FUNCTION_BLOCK FB_TCMultiLevelSeq EXTENDS Tc3_HBI_System.FB_Basic
VAR_INPUT
	iLevel								: UINT;
	lvlAlmMod							: ST_AlarmModules;
END_VAR
VAR_OUTPUT
END_VAR
VAR	
	// Cylinder instance
	fbTCDrawerExtRet					: Tc3_HBI_Cylinder.FB_Cylinder;
	inTCDrawerExtRet					: Tc3_HBI_Cylinder.I_Cylinder:= fbTCDrawerExtRet;
		                        		
	fbTCDrawerUpDn						: Tc3_HBI_Cylinder.FB_Cylinder;
	inTCDrawerUpDn						: Tc3_HBI_Cylinder.I_Cylinder:= fbTCDrawerUpDn;
	
	fbMotor_Ready 						: Tc3_HBI_Utilities.FB_SensorSignal;
	fbMotor_Home_Position 				: Tc3_HBI_Utilities.FB_SensorSignal;
	fbMotor_Position_Reached			: Tc3_HBI_Utilities.FB_SensorSignal;
	fbMotor_Ps_Table_Active				: Tc3_HBI_Utilities.FB_SensorSignal; //temp use for level1 movein ready
	fbMotor_Error						: Tc3_HBI_Utilities.FB_SensorSignal;
	fbBD_ipBdoor 						: Tc3_HBI_Utilities.FB_BackDoor_Digital;
	
	delay								: FB_Delay;
	
	inPOn								: BOOL;
	outPon								: BOOL;

	doorLockChkTim						: TON; // Timer To Check DoorLockFeedBack After DoorLock Output is On.
	
	DIFU								: R_TRIG;
	
	stMLVIO 							: ST_TCMultiLevel_VIO;
	stDbStnVIO							: ST_DebugStation_VIO; // For Debug Sation VIO; 
	stMLDIO 							: ST_TCMultiLevel_DIO;
	stMLBIO								: ST_TCMultiLevel_BIO;
	stTCMLSeqParam 						: ST_TCMultiLevelSeqParam;
	stTCColVIO							: ST_TCColumn_VIO;
	stTCColDIO							: ST_TCColumn_DIO;
	
	//for log purpose
	stOldMLVIO 							: ST_TCMultiLevel_VIO;
	stOldAlarm							: ST_AlarmModules;
	
	FB_M_nCyclic_tSensorDelay			: TIME	:= T#200MS; // By default
	FB_M_nCyclic_tSensorTimeOut			: TIME	:= T#10S;

	// Common var 
	bPause 								: BOOL; // Sequence pause
	bBypassSingleMove 					: BOOL	:= TRUE;
	bStep								: BOOL;
	rtStep								: R_TRIG;
	rtStepCase							: R_TRIG;
	rtError								: R_TRIG;
	iStkSeqCase 						: INT;
	iSeqStep							: INT;
	iSysRsetSeqStep						: INT;
	arrSeqStep							: ARRAY [0..50] OF E_SeqSts; // Seq
	arrSysRsetSeqStep					: ARRAY [0..50] OF E_SeqSts; // Sys Rset seq
	
	sMessage 							: STRING;
	bErrClear							: BOOL;
	bStepDone							: BOOL;
	bSafeExecute						: BOOL;
	iStkSingStackUp						: INT;
	iLibrySts 							: ARRAY [1..20] OF UDINT;
	                            		
	sMsg 								: STRING;
	FB_M_nCyclic_tDelay					: TIME	:= T#200MS;
	
	nI									: UINT;
	rtStartTrig							: R_Trig;
	rtStopTrig							: R_Trig;
	StartPbDly							: Ton;
	StopPbDly							: Ton;
	                            		
	btest								: BOOL;
	
	tDPSDelayToComplete					: TON; // DPSPowerOnOff
	tDPSDelayToAutoComplete				: TON; // DPSPowerAuto
	                            		
	tAPACPwrDelayToComplete				: TON; // AP240ACPowerOnOff
	tAPACPwrDelayToAutoComplete			: TON; // AP240ACPowerAuto
	
	tBef								: TIME; // Before Dwr Action
	tAft								: TIME; // After Dwr Action
	tSpn								: REAL; // Duration Time Span
	tUpDnlock							: BOOL;
	tInOutlock							: BOOL;
	i									: INT;
	pwrOnChkTim							: TON; // PowerOnFeedBackCheck Delay After Power On Durin SystemRset
	
	DIFUTstPresent						: R_TRIG;
	DIFUOn_TstPwr						: R_TRIG;
	DIFUAPPresent						: R_TRIG;
	DIFUOn_AP240Pwr						: R_TRIG;
	DIFUSet_bChkTstOn					: R_TRIG; 	
	DIFUSet_bChkAP240On					: R_TRIG; 	
	
	
	tstOnCheckTim						: TON; // delay to check TesterOnFeedback
	ap240OnCheckTim						: TON; // delay to check AP240OnFeedback
	tstPresentTim						: TON; // delay to On Tester Air Valve after Tester Present
	apPresentTimer						: TON;
	isLeakage							: BOOL;
	isGroundFault						: BOOL;
	isTstPwrOnFault						: BOOL;
	TBOT_TC_ACPower_Signal					: BOOL;
	bTIISenSimArray						: ARRAY[1..NO_OF_TII_SENSOR] OF BOOL;  //TII Sensor Sim by HMI
	bBtnSimArray						: ARRAY[1..NO_OF_BTNLED] OF BOOL;  //Btn Press Sim by HMI

//<TII Interlock>
	itl_opAP_240ACPwrEnable  			: BOOL	:= FALSE;
    itl_opDoorOpenReqLED				: BOOL	:= FALSE;
    itl_opAlarmLED 						: BOOL	:= FALSE;
    itl_opTesterAPDetachReqBtnLED		: BOOL	:= FALSE;
    itl_opTesterDrawerAirOffReqBtnLED   : BOOL	:= FALSE;
    itl_opAP_SafeToMoveSignal           : BOOL	:= FALSE;
    itl_opAP_TCCReset					: BOOL	:= FALSE;
    itl_opCell_LTIMValve				: BOOL	:= FALSE;
    itl_opCellDrawerCylExtend 			: BOOL	:= FALSE;
    itl_opCellDrawerCylRetract 			: BOOL	:= FALSE;
    itl_opCellDrawerCylUp 				: BOOL	:= FALSE;
    itl_opCellDrawerCylDown 			: BOOL	:= FALSE;
    itl_opTst240VACPwrEnable 			: BOOL	:= FALSE;
    itl_opCellPCWValve  				: BOOL	:= FALSE;
    itl_opTIUSktAirSol_1				: BOOL	:= FALSE;
    itl_opTIUSktAirSol_2				: BOOL	:= FALSE;
    itl_opAP_AirSupplySol				: BOOL	:= FALSE;
    itl_opTesterDrawerAirSupplySol	    : BOOL	:= FALSE;
    itl_opCell_24VPowerEnable			: BOOL	:= FALSE;
    itl_opCellDoorClosed				: BOOL	:= FALSE;
	isAboveCellLeakage					: BOOL;
//</TII Interlock>	

//<AirOnOff>
	iAPAirStep							: INT	:= 1;
	iTstAirStep							: INT	:= 1;
	iTIUSktAirStep						: INT	:= 1;
//</AirOnOff>

//<PowerOnOff>
	iAPPwrStep							: INT	:= 1;
	iTstPwrStep							: INT	:= 1;
//</AirOnOff>

	FB_TC_AP240ACPower					: DFB_Cylinder;
	DUT_TC_AP240ACPower					: DUT_Cylinder;
	TC_AP240Power_Perm					: WORD;
	TC_AP240Power_SD					: WORD;
	TC_AP240ACPower_Reset				: R_TRIG;
	TC_AP240ACPower_Precondition		: BOOL; 
	
	FB_opCell24VPowerEnable				: DFB_Cylinder;
	DUT_opCell24VPowerEnable				: DUT_Cylinder;
	Alarm_opCell24VPowerEnable			: BOOL;
	Precondition_opCell24VPowerEnable	: BOOL;
	Reset_opCell24VPowerEnable			: R_TRIG;
	
	TC_APAirSupplySol_Reset				: R_TRIG;
	TC_TesterDrawerAirSupplySol_Reset	: R_TRIG;
END_VAR

METHOD AirOnOff : UDINT
VAR_INPUT
END_VAR
CASE iAPAirStep OF
	1: 	//ON
		//apPresentTimer(IN:=stMLVIO.ipAPPresentSensor, PT:=APPrstChkDelay);
		TC_APAirSupplySol_Reset(CLK:= (NOT itl_opAP_AirSupplySol));
		IF (stMLVIO.bEnableAPAirSupOnInit OR stMLVIO.eAPAirSupCmd=E_Pwr.ON OR TC_APAirSupplySol_Reset.Q) THEN //OR stMLVIO.ipAPReady) (*AND apPresentTimer.Q*) THEN //tytier2
			stMLVIO.opAPAirSupplySol:= TRUE;
		END_IF
		iAPAirStep:=2;
	2:	//ON
		IF stMLVIO.opAPAirSupplySol AND stMLVIO.bEnableAPAirSupOnInit THEN
			stMLVIO.bEnableAPAirSupOnInit:= FALSE;
		END_IF
		iAPAirStep:=3;
	3:	//ON
		IF stMLVIO.opAPAirSupplySol AND stMLVIO.eAPAirSupCmd=E_Pwr.ON THEN
				stMLVIO.eAPAirSupCmd:=E_Pwr.DONE;
		END_IF
		iAPAirStep:=4;
	4:  //OFF
		IF stMLVIO.opAPAirSupplySol
		AND(stMLVIO.eAPAirSupCmd=E_Pwr.OFF OR itl_opAP_AirSupplySol) THEN
		 	stMLVIO.opAPAirSupplySol:= FALSE;
			//stMLVIO.eAPAirSupCmd:=E_Pwr.DONE;
		END_IF
		iAPAirStep:=5;
	5:	//OFF
		IF NOT stMLVIO.opAPAirSupplySol AND stMLVIO.eAPAirSupCmd=E_Pwr.OFF THEN
			stMLVIO.eAPAirSupCmd:=E_Pwr.DONE;
		END_IF
		iAPAirStep:=1;
END_CASE

CASE iTstAirStep OF
	1: 	//ON
		//tstPresentTim(IN:=stMLVIO.ipTesterPresent, PT:=TstPrstChkDelay);
		TC_TesterDrawerAirSupplySol_Reset(CLK:= (NOT itl_opTesterDrawerAirSupplySol));
		IF ( stMLVIO.bEnableDwrAirSupOnInit OR stMLVIO.eTstAirSupCmd=E_Pwr.ON OR TC_TesterDrawerAirSupplySol_Reset.Q) (*AND tstPresentTim.Q*) THEN
			stMLVIO.opTesterDrawerAirSupplySol:= TRUE;
		END_IF
		iTstAirStep:=2;
	2:	//ON
		IF stMLVIO.opTesterDrawerAirSupplySol AND stMLVIO.bEnableDwrAirSupOnInit THEN
			stMLVIO.bEnableDwrAirSupOnInit:= FALSE;
		END_IF
		iTstAirStep:=3;
	3:	//ON
		IF stMLVIO.opTesterDrawerAirSupplySol AND stMLVIO.eTstAirSupCmd=E_Pwr.ON THEN
			stMLVIO.eTstAirSupCmd:=E_Pwr.DONE;
		END_IF
		iTstAirStep:=4;
	4:  //OFF
		iTstAirStep:=5;
	5:	//OFF
		IF 	stMLVIO.opTesterDrawerAirSupplySol 
			AND (stMLVIO.eTstAirSupCmd=E_Pwr.OFF  OR itl_opTesterDrawerAirSupplySol) THEN
			stMLVIO.opTesterDrawerAirSupplySol:= FALSE;
			//stMLVIO.eTstAirSupCmd:=E_Pwr.DONE;
		END_IF
		iTstAirStep:=6;
	6:	//OFF
		IF NOT stMLVIO.opTesterDrawerAirSupplySol AND stMLVIO.eTstAirSupCmd=E_Pwr.OFF THEN
			stMLVIO.eTstAirSupCmd:=E_Pwr.DONE;
		END_IF
		iTstAirStep:=1;
END_CASE

CASE iTIUSktAirStep OF
	1: 	
		iTIUSktAirStep:=2;
	2:
		//ON
		IF NOT stMLVIO.opTIUSktAirSol_1 AND stMLVIO.eTIUSktAir1Cmd=E_Pwr.ON THEN 
			stMLVIO.opTIUSktAirSol_1:= TRUE;
		END_IF
		IF NOT	stMLVIO.opTIUSktAirSol_2 AND stMLVIO.eTIUSktAir2Cmd=E_Pwr.ON THEN
			stMLVIO.opTIUSktAirSol_2:= TRUE;
		END_IF
		iTIUSktAirStep:=3;
		
	3:	//ON
		IF stMLVIO.opTIUSktAirSol_1 AND stMLVIO.eTIUSktAir1Cmd=E_Pwr.ON THEN
			stMLVIO.eTIUSktAir1Cmd:=E_Pwr.DONE;
		END_IF
		IF stMLVIO.opTIUSktAirSol_2 AND stMLVIO.eTIUSktAir2Cmd=E_Pwr.ON THEN
			stMLVIO.eTIUSktAir2Cmd:=E_Pwr.DONE;
		END_IF
		iTIUSktAirStep:=4;
	4:	//OFF
		IF 	stMLVIO.opTIUSktAirSol_1 AND stMLVIO.eTIUSktAir1Cmd=E_Pwr.OFF THEN 
			stMLVIO.opTIUSktAirSol_1:= FALSE;
		END_IF
		IF 	stMLVIO.opTIUSktAirSol_2 AND stMLVIO.eTIUSktAir2Cmd=E_Pwr.OFF THEN 
			stMLVIO.opTIUSktAirSol_2:= FALSE;
		END_IF
		iTIUSktAirStep:=5;
	5:	//OFF
		IF NOT stMLVIO.opTIUSktAirSol_1 AND stMLVIO.eTIUSktAir1Cmd=E_Pwr.OFF THEN
			stMLVIO.eTIUSktAir1Cmd:=E_Pwr.DONE;
		END_IF
		IF NOT stMLVIO.opTIUSktAirSol_1 AND stMLVIO.eTIUSktAir1Cmd=E_Pwr.OFF THEN
			stMLVIO.eTIUSktAir1Cmd:=E_Pwr.DONE;
		END_IF
		
		iTIUSktAirStep:=1;
END_CASE
END_METHOD

METHOD DwrAirOnInit : BOOL
VAR_INPUT
END_VAR
IF NOT stMLVIO.bEnableDwrAirSupOnInit THEN stMLVIO.bEnableDwrAirSupOnInit:=TRUE; END_IF
END_METHOD

METHOD M_240APPwr : UDINT
VAR_INPUT
	iLevel:INT;
END_VAR

//<APPowerOn>
(*	DIFUAPPresent(clk:=stMLVIO.ipAPPresentSensor AND (NOT itl_opAP_240ACPwrEnable));
	IF DIFUAPPresent.Q THEN
		stMLVIO.bAP240ACPowerOnOff 						:= TRUE;
	END_IF

	//OnPower===========================================================================================================
	//TII AP240 PowerOnError
	stMLVIO.bTIIAP240OnError := ALMTC.Level[iLevel].ALarmID[E_TIIAlarm.ipAPPowerOn] 	;
	stMLVIO.bTIIAPPrstError:= ALMTC.Level[iLevel].ALarmID[E_TIIAlarm.ipAPPresentSensor] 	;
	DIFUOn_AP240Pwr(clk:=(stMLVIO.ipAPPresentSensor) AND NOT isLeakage AND NOT isGroundFault AND (stMLVIO.bAP240ACPowerOnOff OR stMLVIO.bEnableAPPwrSupOnInit));
	
	IF DIFUOn_AP240Pwr.Q THEN
		stMLVIO.opAP240ACPwrEnable						:=TRUE;
	END_IF
	ap240OnCheckTim(IN:=stMLVIO.opAP240ACPwrEnable,PT:=APPwrOnChkDelay);
	DIFUSet_bChkAP240On(CLK:=stMLVIO.ipAPPresentSensor AND (stMLVIO.bAP240ACPowerOnOff OR stMLVIO.bEnableAPPwrSupOnInit) AND ap240OnCheckTim.Q);
	IF DIFUSet_bChkAP240On.Q THEN
		//ap240OnCheckTim(IN:=FALSE);
		stMLVIO.bChkAP240On								:=TRUE;	
	END_IF
	//CheckTesterAfter2s=====================================================================================================
	IF (NOT stMLVIO.ipAPPowerOn OR NOT stMLVIO.ipAPPresentSensor)
		AND stMLVIO.bChkAP240On AND stMLVIO.bAP240ACPowerOnOff AND (stMLVIO.bTIIAP240OnError OR stMLVIO.bTIIAPPrstError)THEN
		stMLVIO.bChkAP240On								:=FALSE;
		stMLVIO.opAP240ACPwrEnable						:=FALSE;
		stMLVIO.bAP240ACPowerOnOff						:=FALSE;
		stMLVIO.bEnableAPPwrSupOnInit					:=FALSE;
	END_IF	
	
	//PCW Valve ==============================================================================================================
	IF stMLVIO.ipAPPresentSensor (*AND stMLVIO.bChkAP240On AND stMLVIO.opAP240ACPwrEnable*)AND 
							   NOT  stMLVIO.bTIIAP240OnError AND NOT isLeakage AND NOT isGroundFault 
							   AND NOT (stMLVIO.ipTesterPresent AND NOT stMLVIO.ipTesterPowerOn)
								THEN
		stMLVIO.opCellPCWValve							:=TRUE;
	//ELSIF (*NOT stMLVIO.ipTesterPowerOn*)ALMTC.Level[iLevel].ALarmID[E_TIIAlarm.ipTesterPowerOn]  AND stMLVIO.bChkTesterOn AND stMLVIO.opTst240VACPwrEnable THEN
	//	stMLVIO.opCellPCWValve:=FALSE;
	//	stMLVIO.bChkTesterOn:=FALSE;	
	//	stMLVIO.bDPSPowerOnOff:=FALSE;
	END_IF	
	
	//OFF if Power Off Command ===============================================================================================
	IF NOT stMLVIO.bAP240ACPowerOnOff 	AND NOT stMLVIO.bEnableAPPwrSupOnInit
										AND (stMLVIO.bChkAP240On OR stMLVIO.opAP240ACPwrEnable) THEN
		stMLVIO.bChkAP240On								:=FALSE;				
		stMLVIO.opAP240ACPwrEnable						:=FALSE;
	END_IF
	
	//Off All Output If Leakage
	IF isLeakage OR isGroundFault OR ( NOT stMLVIO.ipAPPresentSensor ) OR (NOT TBOT_TC_ACPower_Signal) OR 
	ALMTC.Level[iLevel].AlarmID[E_TIIAlarm.ipTesterPowerOn]	OR 	eapShutOffAllACPower
	THEN
		stMLVIO.bChkAP240On								:=FALSE;
		stMLVIO.opAP240ACPwrEnable						:=FALSE;
		stMLVIO.bAP240ACPowerOnOff						:=FALSE;
		stMLVIO.bEnableAPPwrSupOnInit					:=FALSE;
		IF (NOT stMLVIO.ipTesterPresent AND NOT stMLVIO.ipAPPresentSensor) OR isLeakage OR isGroundFault THEN
			stMLVIO.opCellPCWValve						:=FALSE;
		END_IF
	END_IF

	//Reset PwrOnInit after Actual power is On
	IF stMLVIO.bEnableAPPwrSupOnInit AND stMLDIO.opAP240ACPwrEnable THEN
		stMLVIO.bEnableAPPwrSupOnInit					:=FALSE;
	END_IF
*)
	
	
	
// new implementation motor
PermSD();

TC_AP240ACPower_Precondition		:= (
											stMLVIO.ipAPPresentSensor AND stMLVIO.ipAPReady	AND	//precondition
											(NOT itl_opAP_240ACPwrEnable) AND 					//TIIAlarm interlock checking
											(NOT DS_Facility_eapShutOffAllACPower OR NOT bDebugCart) AND	//EAP shut off from debug station facility. 1: shutoff, 0: Normal
											(NOT TBOT_TC_ACPower_Signal OR bDebugCart)				//TBOT signal to TC. 1:shutoff, 0: Normal
										) AND			
										stMLVIO.bAP240ACPowerOnOff;								//power on and off manual command);

TC_AP240ACPower_Reset(CLK:= TC_AP240ACPower_Precondition);

DUT_TC_AP240ACPower.AutInp		:= TC_AP240ACPower_Precondition;
DUT_TC_AP240ACPower.Reset		:= TC_AP240ACPower_Reset.Q;
DUT_TC_AP240ACPower.Travel_Time	:= 2;


FB_TC_AP240ACPower(
	Sec_P		:= Sec_P, 
	ID		:= 'TC_AP240ACPower', 
	Simulate		:= DUT_TC_AP240ACPower.Simulate, 
	Permissive		:= TC_AP240Power_Perm, 
	ShutDown		:= TC_AP240Power_SD, 
	AutoInp		:= DUT_TC_AP240ACPower.AutInp, 
	Command		:= DUT_TC_AP240ACPower.CMD, 
	IExtend		:= stMLVIO.ipAPPowerOn, 
	IRetract		:= (NOT stMLVIO.ipAPPowerOn), 
	Travel_Time		:= DUT_TC_AP240ACPower.Travel_Time, 
	SetOutput_Pulse		:= FALSE, 
	FailedHoldLast		:= FALSE,
	OExtend		=> stMLVIO.opAP240ACPwrEnable, 
	ORetract		=> , 
	DUT		:= DUT_TC_AP240ACPower);
//</APPowerOn>

GVL_DUT_TC_AP240ACPower		:= DUT_TC_AP240ACPower;
END_METHOD

METHOD M_240TstPwr : UDINT
VAR_INPUT
	iLevel:INT:=1;
END_VAR
	
//<TesterPowerOn>
	//On Output if Tester Present and DPSPowerOn
	//stMLVIO.opTst240VACPwrEnable 	:=	stMLVIO.bDPSPowerOnOff AND stMLVIO.ipTesterPresent	;
	//TII Tester PowerOnError
	
	stMLVIO.bTIITstPrstError:= ALMTC.Level[iLevel].ALarmID[E_TIIAlarm.ipTesterPresent] 	;
	stMLVIO.bTIITesterOnError := ALMTC.Level[iLevel].ALarmID[E_TIIAlarm.ipTesterPowerOn] 	;
	(*stMLVIO.bTIITesterLatchClosedError := ALMTC.Level[iLevel].ALarmID[E_TIIAlarm.ipTesterLatchesClosed] 	;*)
	//Reset DPSPowerONOFF bit if Tester On Error
	//stMLVIO.bDPSPowerOnOff := NOT stMLVIO.bTIITesterOnError;
	
	//SelfStartForTstPwrOn====================================================================================================
	DIFUTstPresent(clk:=stMLVIO.ipTesterPresent AND stMLVIO.ipTesterLatchesClosed AND (NOT itl_opTst240VACPwrEnable));
	//DIFUTstPresent(clk:=stMLVIO.ipTesterPresent AND stMLVIO.ipTesterLatchesClosed AND NOT stMLVIO.opAlarmLED);//To Auto On After Any Of the Alarm Occurance)
	IF DIFUTstPresent.Q THEN
		stMLVIO.bDPSPowerOnOff := TRUE;
	END_IF
	
	//OnTesterPower===========================================================================================================
	DIFUOn_TstPwr(clk:=stMLVIO.ipTesterPresent AND stMLVIO.ipTesterLatchesClosed AND (stMLVIO.bDPSPowerOnOff OR stMLVIO.bEnableTstPwrSupOnInit));
	IF DIFUOn_TstPwr.Q THEN                                                                                     
		stMLVIO.opTst240VACPwrEnable:=TRUE;
	END_IF
	//TesterOnFeedBackCheckDelay==============================================================================================
	tstOnCheckTim(IN:=stMLVIO.opTst240VACPwrEnable,PT:=TstPwrOnChkDelay); //Wait for 20s after TesterPwr On
	DIFUSet_bChkTstOn(CLK:=stMLVIO.ipTesterPresent	 AND (stMLVIO.bDPSPowerOnOff OR stMLVIO.bEnableTstPwrSupOnInit) AND tstOnCheckTim.Q);
	IF DIFUSet_bChkTstOn.Q THEN
		//tstOnCheckTim(IN:=FALSE);
		stMLVIO.bChkTesterOn:=TRUE;	
	END_IF
	//ResetTimerForNextShot
	//IF stMLVIO.bDPSPowerOnOff AND stMLVIO.bChkTesterOn THEN
	//	tstOnCheckTim(IN:=FALSE);
	//END_IF
	//CheckTesterAfter20s=====================================================================================================
	IF (NOT stMLVIO.ipTesterPowerOn (*OR NOT stMLVIO.ipTesterPresent*) OR NOT stMLVIO.ipTesterLatchesClosed ) 
									AND stMLVIO.bChkTesterOn (*AND stMLVIO.bDPSPowerOnOff *)
									AND (stMLVIO.bTIITesterOnError (*OR stMLVIO.bTIITesterLatchClosedError*) OR stMLVIO.bTIITstPrstError)THEN
		stMLVIO.bChkTesterOn:=FALSE;
		stMLVIO.opTst240VACPwrEnable:=FALSE;
		stMLVIO.bDPSPowerOnOff:=FALSE;
		stMLVIO.opCellPCWValve:=FALSE;
		stMLVIO.bEnableTstPwrSupOnInit:=FALSE;
	END_IF	
	//OFF if Power Off Command ===============================================================================================
	IF NOT stMLVIO.bDPSPowerOnOff AND NOT stMLVIO.bEnableTstPwrSupOnInit 
	   							  AND (stMLVIO.bChkTesterOn OR stMLVIO.opTst240VACPwrEnable   (* OR 
stMLVIO.opCellPCWValve*) )THEN
		stMLVIO.bChkTesterOn:=FALSE;
		stMLVIO.opTst240VACPwrEnable:=FALSE;
		(*stMLVIO.opCellPCWValve:=FALSE;*)
	END_IF
	//PCW Valve ==============================================================================================================

	IF stMLVIO.ipTesterPowerOn AND stMLVIO.bChkTesterOn AND stMLVIO.opTst240VACPwrEnable AND 
							   NOT  stMLVIO.bTIITesterOnError AND NOT isLeakage AND NOT isGroundFault THEN
		stMLVIO.opCellPCWValve:=TRUE;
	//ELSIF (*NOT stMLVIO.ipTesterPowerOn*)ALMTC.Level[iLevel].ALarmID[E_TIIAlarm.ipTesterPowerOn]  AND stMLVIO.bChkTesterOn AND stMLVIO.opTst240VACPwrEnable THEN
	//	stMLVIO.opCellPCWValve:=FALSE;
	//	stMLVIO.bChkTesterOn:=FALSE;	
	//	stMLVIO.bDPSPowerOnOff:=FALSE;
	END_IF	
	//OffPCWValve and All Output If Leakage
	IF isLeakage OR isGroundFault OR ( NOT stMLVIO.ipTesterPresent ) OR TBOT_TC_ACPower_Signal OR DS_Facility_eapShutOffAllACPower THEN
		stMLVIO.bChkTesterOn:=FALSE;	
		stMLVIO.opTst240VACPwrEnable:=FALSE;
		stMLVIO.bDPSPowerOnOff:=FALSE;
		stMLVIO.bEnableTstPwrSupOnInit:=FALSE;
	END_IF
	IF (NOT stMLVIO.ipTesterPresent AND NOT stMLVIO.ipAPPresentSensor) OR isLeakage OR isGroundFault OR
		(stMLVIO.ipTesterPresent AND NOT stMLVIO.ipTesterPowerOn  AND NOT stMLVIO.ipTesterLatchesClosed ) 
	THEN
		stMLVIO.opCellPCWValve:=FALSE;
	END_IF
	
	//Reset PweOnInit after Actual power is On
	IF stMLVIO.bEnableTstPwrSupOnInit AND stMLDIO.opTst240VACPwrEnable THEN
		stMLVIO.bEnableTstPwrSupOnInit:=FALSE;
	END_IF
	//==============================================================================================================
//</TesterPowerOn>
END_METHOD

METHOD M_AboveLeakageChecking : BOOL
VAR_INPUT
	currentLevel	: INT;
END_VAR
VAR
	maxLevel		: INT;
END_VAR
maxLevel									:= NO_OF_LEVEL;

IF currentLevel = maxLevel THEN
	M_AboveLeakageChecking						:= FALSE;
	RETURN;
END_IF

IF ALMTC.Level[currentLevel+1].AlarmID[E_TIIAlarm.ipCellFluidLeakage1] OR ALMTC.Level[currentLevel+1].AlarmID[E_TIIAlarm.ipCellFluidLeakage2] THEN
	M_AboveLeakageChecking					:= TRUE;
ELSIF ALMTC.Level[currentLevel+2].AlarmID[E_TIIAlarm.ipCellFluidLeakage1] OR ALMTC.Level[currentLevel+2].AlarmID[E_TIIAlarm.ipCellFluidLeakage2] THEN
	M_AboveLeakageChecking					:= TRUE;
END_IF
END_METHOD

METHOD M_APSanityCheck : INT
VAR_INPUT
	stMultiLevelVIO	: ST_TCMultiLevel_VIO;
	//stColVIO		: ST_TCCOLUMN_VIO;
END_VAR
VAR_IN_OUT
	sMsg		:STRING;
END_VAR
(*IF (NOT stMultiLevelVIO.ipTCCellDoorOpenCloseStatus) THEN
	sMsg:='Door Closed Signal not Detected Error';
	M_IsSanityCheckFailed									:= E_AlarmID.DoorCloseSignalNotDetected;//31;
ELSIF (NOT stMultiLevelVIO.ipTCCellDoorClosed) THEN
	sMsg:='Door Locked Signal not Detected Error';
	M_IsSanityCheckFailed									:= E_TIIAlarm.ipTCCellDoorClosed;//12;
END_IF

IF bDebugCart THEN 
	IF (NOT stMultiLevelVIO.ipTCCellTbotSideDoorOpenCloseStatus01) THEN
		sMsg:='Front Door Closed_1 Signal not Detected Error';
		M_IsSanityCheckFailed									:= E_AlarmID.TBotSideDoorCloseSignalNotDetected;//33;
	ELSIF (NOT stMultiLevelVIO.ipTCCellTbotSideDoorOpenCloseStatus02) THEN
		sMsg:='Front Door Closed_2 Signal not Detected Error';
		M_IsSanityCheckFailed									:= E_AlarmID.TBotSideDoorCloseSignalNotDetected;//33;
	ELSIF (NOT stMultiLevelVIO.ipTCCellTbotSideDoorLocked01) THEN
		sMsg:='Front Door Lock_1 Signal not Detected Error';
		M_IsSanityCheckFailed									:= E_TIIAlarm.FrontDoorLockSignalNotDetected;//34;
	ELSIF (NOT stMultiLevelVIO.ipTCCellTbotSideDoorLocked02) THEN
		sMsg:='Front Door Lock_2 Signal not Detected Error';
		M_IsSanityCheckFailed									:= E_TIIAlarm.FrontDoorLockSignalNotDetected;//34;
	END_IF
END_IF *)

//Check AP Up
IF stMultiLevelVIO.ipAPPresentSensor THEN
	IF (NOT stMultiLevelVIO.ipHandlerSafeToEnterHwr) OR (NOT stMultiLevelVIO.ipHandlerSafeToEnterPLC) THEN
		sMsg												:= 'AP is not Deactuated (UP)';
		M_APSanityCheck										:= E_AlarmID.APIsNotInUPPosition; //30;
	ELSIF (NOT stMultiLevelVIO.ipAPReady) THEN
		sMsg												:= 'AP is not Ready';
		M_APSanityCheck										:= E_TIIAlarm.ipAPReady; //3;
	END_IF
END_IF
END_METHOD

METHOD M_GetTIUStatus : INT
VAR_INPUT
	b0:BOOL;
	b1:BOOL;
	b2:BOOL;
	b3:BOOL;
END_VAR
VAR
	result:INT;
END_VAR
result.0				:= b0;
result.1				:= b1;
result.2				:= b2;
result.3				:= b3;
M_GetTIUStatus			:= result;
END_METHOD

METHOD M_InitializeCommand : INT
VAR_INPUT
END_VAR
VAR
	stColVIO:ST_TCColumn_VIO;
	isError:BOOL;
	sError:STRING;
	iTIUStatus: INT;
END_VAR
M_InitializeCommand								:= iStkSingStackUp;

IF bPause THEN
	RETURN;
END_IF

IF iSysRsetSeqStep > 0 THEN
	;//Do nothing;
ELSIF stTCMLSeqParam.bInitialise THEN
	arrSysRsetSeqStep[0]										:= E_SeqSts.eInit;
	arrSysRsetSeqStep[1]										:= E_SeqSts.eSanityCheck;
	arrSysRsetSeqStep[2]										:= E_SeqSts.ePwrOn;
	arrSysRsetSeqStep[3]										:= E_SeqSts.eChkTIUPosition;
	arrSysRsetSeqStep[4]										:= E_SeqSts.eTBotEAPSanityCheck;
	arrSysRsetSeqStep[5]										:= E_SeqSts.eMoveDrawerUp;
	arrSysRsetSeqStep[6]										:= E_SeqSts.eTBotEAPSanityCheck;
	arrSysRsetSeqStep[7]										:= E_SeqSts.eMoveDrawerIn;
	arrSysRsetSeqStep[8]										:= E_SeqSts.eMoveDrawerDown;
	arrSysRsetSeqStep[9]										:= E_SeqSts.eDone;
END_IF

//Sequence start
iStkSeqCase									:= arrSysRsetSeqStep[iSysRsetSeqStep];

// State machine
CASE iStkSeqCase OF
	E_SeqSts.eInit:
		
		sMessage										:=' Start Executing';
		bStepDone										:=TRUE;
		
	E_SeqSts.eSanityCheck:
		sMessage										:= ' Sanity Check';
		_nErrorID										:= INT_TO_UDINT(M_APSanityCheck(
																			stMultiLevelVIO	:= stMLVIO, 
																			sMsg			:= sMessage
																		));
																						
		IF (NOT stMLVIO.ipTCCellDoorOpenCloseStatus) THEN
			sMessage									:= 'Door Closed Signal not Detected Error';
			_nErrorID									:= E_AlarmID.DoorCloseSignalNotDetected;//31;
		ELSIF (NOT stMLVIO.ipTCCellDoorClosed) THEN
			sMessage									:= 'Door Locked Signal not Detected Error';
			_nErrorID									:= E_TIIAlarm.ipTCCellDoorClosed;//12;
		END_IF
		
		IF (NOT bDebugCart) THEN
			// drawer up signal alarm
			IF ALMTC.Level[iLevel].AlarmID[E_TIIAlarm.ipTCDrawerUpSignal] THEN
				sMessage									:= 'Drawer Up Signal not detected';
				_nErrorID									:= E_TIIAlarm.ipTCDrawerUpSignal;
				
			// drawer extend alarm
			ELSIF ALMTC.Level[iLevel].AlarmID[E_TIIAlarm.ipTCDrawerExtendSignal] THEN
				sMessage									:= 'Drawer Extend Signal not detected';
				_nErrorID									:= E_TIIAlarm.ipTCDrawerExtendSignal;
			
			// drawer retract alarm
			ELSIF ALMTC.Level[iLevel].AlarmID[E_TIIAlarm.ipTCDrawerRetractSignal] THEN
				sMessage									:= 'Drawer Retract Signal not detected';
				_nErrorID									:= E_TIIAlarm.ipTCDrawerRetractSignal;
				
			// tester latch alarm	
			ELSIF ALMTC.Level[iLevel].AlarmID[E_TIIAlarm.ipTesterLatchesClosed] THEN
				sMessage									:= 'Tester Latches Signal not detected';
				_nErrorID									:= E_TIIAlarm.ipTesterLatchesClosed;
			END_IF
		END_IF
		
		IF bDebugCart THEN 
			IF (NOT stMLVIO.ipTCCellTbotSideDoorOpenCloseStatus01) THEN
				sMessage									:= 'Front Door Closed_1 Signal not Detected Error';
				_nErrorID									:= E_AlarmID.TBotSideDoorCloseSignalNotDetected;//33;
			ELSIF (NOT stMLVIO.ipTCCellTbotSideDoorOpenCloseStatus02) THEN
				sMessage									:= 'Front Door Closed_2 Signal not Detected Error';
				_nErrorID									:= E_AlarmID.TBotSideDoorCloseSignalNotDetected;//33;
			ELSIF (NOT stMLVIO.ipTCCellTbotSideDoorLocked01) THEN
				sMessage									:= 'Front Door Lock_1 Signal not Detected Error';
				_nErrorID									:= E_TIIAlarm.FrontDoorLockSignalNotDetected;//34;
			ELSIF (NOT stMLVIO.ipTCCellTbotSideDoorLocked02) THEN
				sMessage									:= 'Front Door Lock_2 Signal not Detected Error';
				_nErrorID									:= E_TIIAlarm.FrontDoorLockSignalNotDetected;//34;
			END_IF
		END_IF 																				
																						
		IF _nErrorID=0 THEN
			bStepDone										:= TRUE;
		END_IF
		
	E_SeqSts.eTBotEAPSanityCheck:
	
		sMessage							:= ' Checking TBot EAP';
	
	
		_nErrorID							:= INT_TO_UDINT(M_IsEAPError(sMsg=>sMessage));
		IF _nErrorID=0 THEN
			bStepDone						:= TRUE;
		END_IF
	
	E_SeqSts.eCheckDoorLock:
		
		IF NOT stMLVIO.ipTCCellDoorClosed THEN
			sError							:= 'Door Lock Signal not Detected Error';
		ELSIF NOT stMLVIO.ipTCCellTbotSideDoorLocked01 AND bDebugCart THEN
			sError							:= 'Front Door Lock_1 Signal not Detected Error';
		ELSIF NOT stMLVIO.ipTCCellTbotSideDoorLocked02 AND bDebugCart THEN
			sError							:= 'Front Door Lock_2 Signal not Detected Error';
		END_IF
	
		IF sError<>'' THEN
			sMessage						:= CONCAT(sMessage,sError);
			_bError							:= TRUE;
			bStepDone						:= FALSE;
		ELSE
			bStepDone						:= TRUE;
		END_IF
		
		
	E_SeqSts.ePwrOn:
		sMessage											:= ' Enable Air Supply ';
		M_Pwr(
			e												:= TRUE);
		
		pwrOnChkTim(
			In												:= TRUE,
			PT												:= INT_TO_TIME(1));
		IF pwrOnChkTim.Q THEN
			pwrOnChkTim(In:=FALSE);
			bStepDone										:= TRUE;
		END_IF
	
	eChkTIUPosition:
		iTIUStatus							:= M_GetTIUStatus(
													b3	:= stMLVIO.ipTCDrawerCylUpRS, 		//UP
													b2	:= stMLVIO.ipTCDrawerCylDownRS,	//DOWN
													b1	:= stMLVIO.ipTCDrawerCylExtendRS,	//EXTEND
													b0	:= stMLVIO.ipTCDrawerCylRetractRS	//RETRACT
											);
											
		CASE iTIUStatus OF 
			0:(*UpInDn*)	bStepDone				:= TRUE;
			1:(*Down*)		iSysRsetSeqStep			:= 7;
			2:(*UpInDn*)	bStepDone				:= TRUE;
			3:(*V_Err*)		_nErrorID				:= E_AlarmID.BothTIUUpDownSignalDetected; sMessage:= 'Both Reed Switchs of Cylinder are Detected';
			4:(*UpInDn*)	bStepDone				:= TRUE;
			5:(*Done*)		iSysRsetSeqStep			:= 7;
			6:(*UpInDn*)	bStepDone				:= TRUE;
			7:(*V_Err*)		_nErrorID				:= E_AlarmID.BothTIUUpDownSignalDetected; sMessage:= 'Both Reed Switchs of Cylinder are Detected';
			8:(*UpInDn*)	bStepDone				:= TRUE;
			9:(*Down*)		iSysRsetSeqStep			:= 7;
			10:(*UpInDn*)	bStepDone				:= TRUE;
			11,(*V_Err*)	
			12,(*H_Err*)	
			13,(*H_Err*)	
			14,(*H_Err*)	
			15:(*H_Err*)	_nErrorID				:= E_AlarmID.BothTIUExternRetractSignalDetected; sMessage:= 'Both Reed Switchs of Cylinder are Detected';
		END_CASE
		
	E_SeqSts.eMoveDrawerUp:
		DwrAirOnInit();
		sMessage						:= ' Drawer Up';
		iLibrySts[1]					:= M_nCmptUpDown(
												bExtend			:= TRUE,  
												sErrorMSg		:= sMsg
											);
		
		IF iLibrySts[1]=10 THEN
			bStepDone					:= TRUE;
		ELSIF iLibrySts[1]=99 THEN
			sMessage					:= CONCAT(sMessage,sMsg);
			_bError						:= TRUE;
		END_IF	
		
	E_SeqSts.eMoveDrawerIn:	
		DwrAirOnInit();
		sMessage						:= ' Drawer In ';
		iLibrySts[1]					:= M_nCmptInOut(bExtend:=FALSE,  sErrorMSg:=sMsg);
		IF iLibrySts[1]=10 THEN
			bStepDone					:= TRUE;
		ELSIF iLibrySts[1]=99 THEN
			sMessage					:= CONCAT(sMessage,sMsg);
			_bError						:= TRUE;
		END_IF
		
	E_SeqSts.eMoveDrawerDown:
		DwrAirOnInit();
		sMessage						:= ' Drawer Down';
		iLibrySts[1]					:= M_nCmptUpDown(
											bExtend:=FALSE,  
											sErrorMSg:=sMsg
											);
		
		IF iLibrySts[1]=10 THEN
			bStepDone							:= TRUE;
		ELSIF iLibrySts[1]=99 THEN
			sMessage							:= CONCAT(sMessage,sMsg);
			_bError								:= TRUE;
		END_IF
		
	E_SeqSts.eDone:	
		DwrAirOnInit();	
		sMessage								:= 'Done';
		M_InitializeCommand						:= 10;
END_CASE	


IF _nErrorID>0 OR _bError THEN
	_bError								:= TRUE;
ELSIF (stMLVIO.bStep OR stMLVIO.bBypassSingleMove OR iStkSeqCase<=E_SeqSts.eSanityCheck) AND iStkSeqCase<E_SeqSts.eDone AND bStepDone THEN
	iSysRsetSeqStep						:= iSysRsetSeqStep+1;
END_IF
END_METHOD

METHOD M_InputBackDoor : UDINT
VAR_INPUT
END_VAR
///////////////////////////////////////////////////////////////////////////////////////////////////////////////////////////////////////////////////////////////////////////////////////////////
////////////////////////// HMI_TII_Sensor_Simulation ////////////////////////
///////////////////////////////////////////////////////////////////////////////////////////////////////////////////////////////////////////////////////////////////////////////////////////////	
IF bHMIEnTIISenSimulation THEN
	FOR i:=1 TO NO_OF_TII_SENSOR DO
		bTIISenSimArray[i]				:= NOT stHMITIISenSimArray[iLevel].bHMITIIByPassArray[i];
	END_FOR
ELSE
	FOR i:=1 TO NO_OF_TII_SENSOR DO
		bTIISenSimArray[i]				:= TRUE;
	END_FOR
END_IF

///////////////////////////////////////////////////////////////////////////////////////////////////////////////////////////////////////////////////////////////////////////////////////////////
////////////////////////// HMI_ManualBtnPress_Simulation ////////////////////////
///////////////////////////////////////////////////////////////////////////////////////////////////////////////////////////////////////////////////////////////////////////////////////////////
IF bHMIBtnSimulation THEN
	FOR i:=1 TO NO_OF_BTNLED DO
		bBtnSimArray[i]					:= NOT stHMIBtnSimArray[iLevel].bHMITIIByPassArray[i];
	END_FOR
ELSE
	FOR i:=1 TO NO_OF_BTNLED DO
		bBtnSimArray[i]					:= TRUE;
	END_FOR
END_IF	

///////////////////////////////////////////////////////////////////////////////////////////////////////////////////////////////////////////////////////////////////////////////////////////////
//////////////////////// Input mapping with Production/Simulation Method 													////////////////////////
//////////////////////// IF bProductionMode, TRUE : Method will use Actual IO, FALSE: Method will use Backdoor IO 			////////////////////////
////////////////////////////////////////////////////////////////////////////////////////////////////////////////////////////////////////////////////////////////////////////////////////////////								
stMLVIO.ipAPPresentSensor 					:= fbBD_ipBdoor.M_bBackDoorCtrl(
																bProductionMode			:= bProductionMode AND bTIISenSimArray[E_TIIAlarm.ipAPPresentSensor], 
																bActual					:= stMLDIO.ipAPPresentSensor, 
   																bSimu					:= TRUE, 
																iBackDoor				:= stMLBIO.ipAPPresentSensor);
										                                                   
stMLVIO.ipAPPowerOn							:= fbBD_ipBdoor.M_bBackDoorCtrl(               
																bProductionMode			:= bProductionMode AND bTIISenSimArray[E_TIIAlarm.ipAPPowerOn], 
                                            					bActual					:= stMLDIO.ipAPPowerOn, 
                                            					bSimu					:= TRUE, 
                                            					iBackDoor				:= stMLBIO.ipAPPowerOn);
                                                                                           
stMLVIO.ipAPReady							:= fbBD_ipBdoor.M_bBackDoorCtrl(               
																bProductionMode			:= bProductionMode AND bTIISenSimArray[E_TIIAlarm.ipAPReady], 
                                            					bActual					:= stMLDIO.ipAPReady, 
                                            					bSimu					:= TRUE, 
                                            					iBackDoor				:= stMLBIO.ipAPReady);
			                                                                               
stMLVIO.ipHandlerSafeToEnterPLC				:= fbBD_ipBdoor.M_bBackDoorCtrl(               
																bProductionMode			:= bProductionMode, 
                                            					bActual					:= stMLDIO.ipHandlerSafeToEnterPLC, 
                                            					bSimu					:= TRUE, 
                                            					iBackDoor				:= stMLBIO.ipHandlerSafeToEnterPLC);
                                                                                           
stMLVIO.ipHandlerSafeToEnterHwr				:= fbBD_ipBdoor.M_bBackDoorCtrl(               
																bProductionMode			:= bProductionMode, 
                                            					bActual					:= stMLDIO.ipHandlerSafeToEnterHwr, 
                                            					bSimu					:= TRUE, 
                                            					iBackDoor				:= stMLBIO.ipHandlerSafeToEnterHwr);
		                                                                                   
stMLVIO.ipCellFluidLeakage1					:= NOT fbBD_ipBdoor.M_bBackDoorCtrl(           
																	bProductionMode		:= bProductionMode AND bTIISenSimArray[E_TIIAlarm.ipCellFluidLeakage1], 
                                            						bActual				:= stMLDIO.ipCellFluidLeakage1, 
                                            						bSimu				:= TRUE, 
                                            						iBackDoor			:= stMLBIO.ipCellFluidLeakage1);
			                                                                               
stMLVIO.ipCellFluidLeakage2					:= NOT fbBD_ipBdoor.M_bBackDoorCtrl(           
																	bProductionMode		:= bProductionMode AND bTIISenSimArray[E_TIIAlarm.ipCellFluidLeakage2], 
                                            						bActual				:= stMLDIO.ipCellFluidLeakage2, 
                                            						bSimu				:= TRUE, 
                                            						iBackDoor			:= stMLBIO.ipCellFluidLeakage2);
			                                                                               
stMLVIO.ipCellGroundFault 					:= fbBD_ipBdoor.M_bBackDoorCtrl(               
																bProductionMode			:= bProductionMode AND bTIISenSimArray[E_TIIAlarm.ipCellGroundFault], 
                                            					bActual					:= stMLDIO.ipCellGroundFault, 
                                            					bSimu					:= FALSE, 
                                            					iBackDoor				:= stMLBIO.ipCellGroundFault);
			                                                                               
stMLVIO.ipTesterPresent						:= fbBD_ipBdoor.M_bBackDoorCtrl(               
																bProductionMode			:= bProductionMode AND bTIISenSimArray[E_TIIAlarm.ipTesterPresent], 
                                            					bActual					:= stMLDIO.ipTesterPresent, 
                                            					bSimu					:= TRUE, 
                                            					iBackDoor				:= stMLBIO.ipTesterPresent);
                                                                                           
stMLVIO.ipTesterPowerOn						:= fbBD_ipBdoor.M_bBackDoorCtrl(               
																bProductionMode			:= bProductionMode AND bTIISenSimArray[E_TIIAlarm.ipTesterPowerOn], 
                                            					bActual					:= stMLDIO.ipTesterPowerOn, 
                                            					bSimu					:= TRUE, 
                                            					iBackDoor				:= stMLBIO.ipTesterPowerOn);
                                                                                           
stMLVIO.ipTesterReady						:= fbBD_ipBdoor.M_bBackDoorCtrl(               
																bProductionMode			:= bProductionMode, 
																bActual					:= stMLDIO.ipTesterReady, 
																bSimu					:= TRUE, 
																iBackDoor				:= stMLBIO.ipTesterReady);
																				           
																				           
stMLVIO.ipTCCellDoorOpenReqBtn				:= fbBD_ipBdoor.M_bBackDoorCtrl(               
																bProductionMode			:= bProductionMode AND bBtnSimArray[2+1], 
                                            					bActual					:= stMLDIO.ipTCCellDoorOpenReqBtn, 
                                            					bSimu					:= FALSE, 
                                            					iBackDoor				:= stMLBIO.ipTCCellDoorOpenReqBtn);
                                                                                    	
stMLVIO.ipDrawerMaintenanceModeBtn			:= fbBD_ipBdoor.M_bBackDoorCtrl(        	
																bProductionMode			:= bProductionMode AND bBtnSimArray[0+1], 
                                            					bActual					:= stMLDIO.ipDrawerMaintenanceModeBtn, 
                                            					bSimu					:= FALSE, 
                                            					iBackDoor				:= stMLBIO.ipDrawerMaintenanceModeBtn);
                                                                                    	   
stMLVIO.ipTCCellAbortFlowBtn				:= fbBD_ipBdoor.M_bBackDoorCtrl(        	   
																bProductionMode			:= bProductionMode AND bBtnSimArray[1+1], 
                                            					bActual					:= stMLDIO.ipTCCellAbortFlowBtn, 
                                            					bSimu					:= FALSE, 
                                            					iBackDoor				:= stMLBIO.ipTCCellAbortFlowBtn);																				  
																				  

IF (stMLVIO.bPLCRebootStatusForExtRetRs AND fbTCDrawerExtRet.P_opRetract) OR fbTCDrawerExtRet.P_opExtend THEN
	stMLVIO.bPLCRebootStatusForExtRetRs :=FALSE;
END_IF
IF (stMLVIO.bPLCRebootStatusForUpDownRs AND fbTCDrawerUpDn.P_opRetract) OR fbTCDrawerUpDn.P_opExtend  THEN
	stMLVIO.bPLCRebootStatusForUpDownRs :=FALSE;
END_IF

inTCDrawerExtRet.P_ipExtend:=stMLVIO.ipTCDrawerCylExtendRS		:=fbBD_ipBdoor.M_bBackDoorCtrl(
																					bProductionMode		:= bProductionMode, 
																					bActual				:= stMLDIO.ipTCDrawerCylExtendRS,
																					bSimu				:= fbTCDrawerExtRet.P_opExtend, 
																					iBackDoor			:= stMLBIO.ipTCDrawerCylExtendRS);

inTCDrawerExtRet.P_ipRetract:=stMLVIO.ipTCDrawerCylRetractRS	:= fbBD_ipBdoor.M_bBackDoorCtrl(
																					bProductionMode		:= bProductionMode, 
																					bActual				:= stMLDIO.ipTCDrawerCylRetractRS,
																					bSimu				:= stMLVIO.bPLCRebootStatusForExtRetRs OR fbTCDrawerExtRet.P_opRetract, 
																					iBackDoor			:= stMLBIO.ipTCDrawerCylRetractRS);
                                                                                                           
inTCDrawerUpDn.P_ipExtend:=stMLVIO.ipTCDrawerCylUpRS			:= fbBD_ipBdoor.M_bBackDoorCtrl(	       
																					bProductionMode		:= bProductionMode, 
																					bActual				:= stMLDIO.ipTCDrawerCylUpRS, 
																					bSimu				:= fbTCDrawerUpDn.P_opExtend, 
																					iBackDoor			:= stMLBIO.ipTCDrawerCylUpRS);
																								  
inTCDrawerUpDn.P_ipRetract:=stMLVIO.ipTCDrawerCylDownRS			:= fbBD_ipBdoor.M_bBackDoorCtrl(
																					bProductionMode		:= bProductionMode, 
																					bActual				:= stMLDIO.ipTCDrawerCylDownRS, 
																					bSimu				:= stMLVIO.bPLCRebootStatusForUpDownRs OR fbTCDrawerUpDn.P_opRetract, 
																					iBackDoor			:= stMLBIO.ipTCDrawerCylDownRS);

																			  
stMLVIO.ipTCCellDoorClosed							:= fbBD_ipBdoor.M_bBackDoorCtrl(
																		bProductionMode		:= bProductionMode AND bTIISenSimArray[E_TIIAlarm.ipTCCellDoorClosed], 
																		bActual				:= stMLDIO.ipTCCellDoorClosed, 
																		bSimu				:= stMLDIO.opCellDoorClosed, 
																		iBackDoor			:= stMLBIO.ipTCCellDoorClosed);
																
stMLVIO.ipTCCellTbotSideDoorLocked01				:= fbBD_ipBdoor.M_bBackDoorCtrl(
																		bProductionMode		:= bProductionMode, 
                                            							bActual				:= stMLDIO.ipTCCellTbotSideDoorLocked01, 
                                            							bSimu				:= stMLDIO.opCellTBOtSideDoorClosed1, 
                                            							iBackDoor			:= stMLBIO.ipTCCellTbotSideDoorLocked01);

stMLVIO.ipTCCellTbotSideDoorLocked02				:= fbBD_ipBdoor.M_bBackDoorCtrl(
																		bProductionMode		:= bProductionMode, 
                                            							bActual				:= stMLDIO.ipTCCellTbotSideDoorLocked02, 
                                            							bSimu				:= stMLDIO.opCellTBOtSideDoorClosed2, 
                                            							iBackDoor			:= stMLBIO.ipTCCellTbotSideDoorLocked02);	
																		
stMLVIO.ipTCCellDoorOpenCloseStatus					:= fbBD_ipBdoor.M_bBackDoorCtrl(
																		bProductionMode		:= bProductionMode, 
                                                						bActual				:= stMLDIO.ipTCCellDoorOpenCloseStatus, 
                                                						bSimu				:= TRUE, 
                                                						iBackDoor			:= stMLBIO.ipTCCellDoorOpenCloseStatus);
																	
stMLVIO.ipTCCellTbotSideDoorOpenCloseStatus01		:= fbBD_ipBdoor.M_bBackDoorCtrl(
																		bProductionMode		:= bProductionMode, 
                                            							bActual				:= stMLDIO.ipTCCellTbotSideDoorOpenCloseStatus01, 
                                            							bSimu				:= TRUE, 
                                            							iBackDoor			:= stMLBIO.ipTCCellTbotSideDoorOpenCloseStatus01);

stMLVIO.ipTCCellTbotSideDoorOpenCloseStatus02		:= fbBD_ipBdoor.M_bBackDoorCtrl(
																		bProductionMode		:= bProductionMode, 
                                            							bActual				:= stMLDIO.ipTCCellTbotSideDoorOpenCloseStatus02, 
                                            							bSimu				:= TRUE, 
                                            							iBackDoor			:= stMLBIO.ipTCCellTbotSideDoorOpenCloseStatus02);	
	
stMLVIO.ipTesterLatchesClosed						:= fbBD_ipBdoor.M_bBackDoorCtrl(
																		bProductionMode		:= bProductionMode AND bTIISenSimArray[E_TIIAlarm.ipTesterLatchesClosed], 
                                            							bActual				:= stMLDIO.ipTesterLatchesClosed, 
                                            							bSimu				:= TRUE, 
                                            							iBackDoor			:= stMLBIO.ipTesterLatchesClosed);
	
																		
/////////////////////////////////////////////////////////////////////////////////////////////////////////////////////////////////////////////////////////////////////////////////////////
////////////////////////// Input mapping simulation in VISU //////////////////////////
////////////////////////////////////////////////////////////////////////////////////////////////////////////////////////////////////////////////////////////////////////////////////////
IF (NOT bProductionMode) THEN
	stMLDIO.ipAPPresentSensor							:= stMLVIO.ipAPPresentSensor;
	stMLDIO.ipAPPowerOn									:= stMLVIO.ipAPPowerOn;
	stMLDIO.ipAPReady									:= stMLVIO.ipAPReady;
	stMLDIO.ipHandlerSafeToEnterPLC						:= stMLVIO.ipHandlerSafeToEnterPLC;
	stMLDIO.ipHandlerSafeToEnterHwr						:= stMLVIO.ipHandlerSafeToEnterHwr;
	stMLDIO.ipCellFluidLeakage1							:= NOT stMLVIO.ipCellFluidLeakage1;
	stMLDIO.ipCellFluidLeakage2							:= NOT stMLVIO.ipCellFluidLeakage2;
	stMLDIO.ipCellGroundFault							:= stMLVIO.ipCellGroundFault;
	stMLDIO.ipTesterPresent								:= stMLVIO.ipTesterPresent;
	stMLDIO.ipTesterPowerOn								:= stMLVIO.ipTesterPowerOn;
	stMLDIO.ipTesterReady								:= stMLVIO.ipTesterReady;
	stMLDIO.ipTCCellDoorOpenReqBtn						:= stMLVIO.ipTCCellDoorOpenReqBtn;
	stMLDIO.ipDrawerMaintenanceModeBtn					:= stMLVIO.ipDrawerMaintenanceModeBtn;
	stMLDIO.ipTCCellAbortFlowBtn						:= stMLVIO.ipTCCellAbortFlowBtn;
	stMLDIO.ipTCDrawerCylExtendRS						:= stMLVIO.ipTCDrawerCylExtendRS;
	stMLDIO.ipTCDrawerCylRetractRS						:= stMLVIO.ipTCDrawerCylRetractRS;
	stMLDIO.ipTCDrawerCylUpRS							:= stMLVIO.ipTCDrawerCylUpRS;
	stMLDIO.ipTCDrawerCylDownRS							:= stMLVIO.ipTCDrawerCylDownRS;
	stMLDIO.ipTCCellDoorClosed							:= stMLVIO.ipTCCellDoorClosed;
	stMLDIO.ipTCCellTbotSideDoorLocked01				:= stMLVIO.ipTCCellTbotSideDoorLocked01;
	stMLDIO.ipTCCellTbotSideDoorLocked02				:= stMLVIO.ipTCCellTbotSideDoorLocked02;
	stMLDIO.ipTCCellDoorOpenCloseStatus					:= stMLVIO.ipTCCellDoorOpenCloseStatus;
	stMLDIO.ipTCCellTbotSideDoorOpenCloseStatus01		:= stMLVIO.ipTCCellTbotSideDoorOpenCloseStatus01;
	stMLDIO.ipTCCellTbotSideDoorOpenCloseStatus02		:= stMLVIO.ipTCCellTbotSideDoorOpenCloseStatus02;
	stMLDIO.ipTesterLatchesClosed						:= stMLVIO.ipTesterLatchesClosed;
	
END_IF
END_METHOD

METHOD M_InterlockTII : UDINT
VAR_INPUT
	ilevel:INT;
END_VAR
///////////////////////////////////////////////////////////////////////////////////////////////////////////////////////////////////////////////////////////////////////////////////////////
///////////////// Get Alarm Interlock to shut off logical outputs ///////////////////////////
///////////////////////////////////////////////////////////////////////////////////////////////////////////////////////////////////////////////////////////////////////////////////////////
isAboveCellLeakage				:= M_AboveLeakageChecking(currentLevel:= ilevel);

									
itl_opTst240VACPwrEnable				:=		ALMTC.Level[iLevel].ALarmID[E_TIIAlarm.ipTesterPresent	  	 	]		OR	
												ALMTC.Level[iLevel].ALarmID[E_TIIAlarm.ipTesterPowerOn	   		]		OR	
												ALMTC.Level[iLevel].ALarmID[E_TIIAlarm.ipTesterLatchesClosed 	]		OR	
												ALMTC.Level[iLevel].ALarmID[E_TIIAlarm.ipCellFluidLeakage1		]		OR	
												ALMTC.Level[iLevel].ALarmID[E_TIIAlarm.ipCellFluidLeakage2		]		OR	
												ALMTC.Level[iLevel].ALarmID[E_TIIAlarm.ipCellGroundFault 	   	]		OR	
												ALMTC.Common.AlarmID[E_ColAlarm.ipColumnFluid_PCW_Leakage 		]		OR	
												ALMTC.Level[iLevel].ALarmID[E_TIIAlarm.TBOT_TC_ACPower_Signal 	]		OR	
												ALMTC.Level[iLevel].AlarmID[E_TIIAlarm.DS_Facility_EAP_ACPower_Signal]	OR 	
												isAboveCellLeakage;

itl_opCell_24VPowerEnable				:=		ALMTC.Level[iLevel].ALarmID[E_TIIAlarm.ipCellFluidLeakage1		]	OR	
												ALMTC.Level[iLevel].ALarmID[E_TIIAlarm.ipCellFluidLeakage2		]	OR	
												ALMTC.Level[iLevel].ALarmID[E_TIIAlarm.ipCellGroundFault 	   	]	OR	
												ALMTC.Common.AlarmID[E_ColAlarm.ipColumnFluid_PCW_Leakage 		]	OR 	
												isAboveCellLeakage;		
                                
itl_opAP_240ACPwrEnable					:=		ALMTC.Level[iLevel].ALarmID[E_TIIAlarm.ipTesterPowerOn			]		OR	
												ALMTC.Level[iLevel].AlarmID[E_TIIAlarm.ipAPPowerOn				]		OR 	
												ALMTC.Level[iLevel].ALarmID[E_TIIAlarm.ipAPReady				]		OR	
												ALMTC.Level[iLevel].ALarmID[E_TIIAlarm.ipCellFluidLeakage1		]		OR	
												ALMTC.Level[iLevel].ALarmID[E_TIIAlarm.ipCellFluidLeakage2		]		OR	
												ALMTC.Level[iLevel].ALarmID[E_TIIAlarm.ipCellGroundFault 	   	]		OR	
												ALMTC.Common.AlarmID[E_ColAlarm.ipColumnFluid_PCW_Leakage 		]		OR	
												ALMTC.Level[iLevel].ALarmID[E_TIIAlarm.TBOT_TC_ACPower_Signal 	]		OR	
												ALMTC.Level[iLevel].AlarmID[E_TIIAlarm.DS_Facility_EAP_ACPower_Signal]	OR 	
												isAboveCellLeakage;	
                                
itl_opCellPCWValve						:=		ALMTC.Level[iLevel].ALarmID[E_TIIAlarm.ipTesterPowerOn			]	OR	
												ALMTC.Level[iLevel].ALarmID[E_TIIAlarm.ipCellFluidLeakage1		]	OR	
												ALMTC.Level[iLevel].ALarmID[E_TIIAlarm.ipCellFluidLeakage2		]	OR	
												ALMTC.Level[iLevel].ALarmID[E_TIIAlarm.ipCellGroundFault 	   	]	OR	
												ALMTC.Common.AlarmID[E_ColAlarm.ipColumnFluid_PCW_Leakage 		]	OR 	
												isAboveCellLeakage;	
							
itl_opAP_AirSupplySol					:=		ALMTC.Level[iLevel].ALarmID[E_TIIAlarm.ipCellFluidLeakage1		]	OR	
												ALMTC.Level[iLevel].ALarmID[E_TIIAlarm.ipCellFluidLeakage2		]	OR	
												ALMTC.Level[iLevel].ALarmID[E_TIIAlarm.ipCellGroundFault 	   	]	OR	
												ALMTC.Common.AlarmID[E_ColAlarm.ipColumnFluid_PCW_Leakage 		]	OR	
												ALMTC.Level[iLevel].AlarmID[E_TIIAlarm.ipAPReady				]	OR 	
												isAboveCellLeakage;
                               
itl_opTesterDrawerAirSupplySol			:=		ALMTC.Level[iLevel].ALarmID[E_TIIAlarm.ipCellFluidLeakage1		]	OR	
												ALMTC.Level[iLevel].ALarmID[E_TIIAlarm.ipCellFluidLeakage2		]	OR	
												ALMTC.Level[iLevel].ALarmID[E_TIIAlarm.ipCellGroundFault 	   	]	OR	
												ALMTC.Common.AlarmID[E_ColAlarm.ipColumnFluid_PCW_Leakage 		]	OR 	
												isAboveCellLeakage;	
								
itl_opAP_SafeToMoveSignal				:=		ALMTC.Level[iLevel].AlarmID[E_TIIAlarm.ipTesterLatchesClosed		]	OR
												ALMTC.Level[iLevel].AlarmID[E_TIIAlarm.ipTCDrawerRetractSignal		]	OR
												ALMTC.Level[iLevel].AlarmID[E_TIIAlarm.ipTCDrawerDownSignal			]	OR	
												ALMTC.Level[iLevel].AlarmID[E_TIIAlarm.ipTCCellDoorClosed			]	OR	
												ALMTC.Common.AlarmID[E_ColAlarm.ipTbotDoorClosedSignal				]	OR 	
												ALMTC.Level[iLevel].AlarmID[E_TIIAlarm.ipCellGroundFault 	   		]	OR	
												ALMTC.Level[iLevel].AlarmID[E_TIIAlarm.ipCellFluidLeakage1 	   		] 	OR	
												ALMTC.Level[iLevel].AlarmID[E_TIIAlarm.ipCellFluidLeakage2 	   		]	OR	
												ALMTC.Common.AlarmID[E_ColAlarm.ipColumnFluid_PCW_Leakage			]	OR	
												ALMTC.Level[iLevel].AlarmID[E_TIIAlarm.FrontDoorLockSignalNotDetected]	OR	
												ALMTC.Level[iLevel].AlarmID[E_TIIAlarm.DS_Facility_EAP_ACPower_Signal]	OR	
												ALMTC.Level[iLevel].AlarmID[E_TIIAlarm.TBOT_TC_ACPower_Signal		]	OR 	
												isAboveCellLeakage;
END_METHOD

METHOD M_IOMapping : UDINT
VAR_INPUT
	ilevel:INT;
END_VAR

VAR_IN_OUT
	//dIO : ST_TCMultiLevel_DIO;
	//vIO : ST_TCMultiLevel_VIO;
	//vIO : ST_TCMultiLevel_BIO;
	//stTCMultiLevelSeqParam : ST_TCMultiLevelSeqParam;	
END_VAR
VAR
//	itl_opAP_240ACPwrEnable  			:BOOL:=FALSE;
//    itl_opDoorOpenReqLED				:BOOL:=FALSE;
//    itl_opAlarmLED 						:BOOL:=FALSE;
//    itl_opTesterAPDetachReqBtnLED		:BOOL:=FALSE;
//    itl_opTesterDrawerAirOffReqBtnLED   :BOOL:=FALSE;
//    itl_opAP_SafeToMoveSignal           :BOOL:=FALSE;
//    itl_opAP_TCCReset					:BOOL:=FALSE;
//    itl_opCell_LTIMValve				:BOOL:=FALSE;
//    itl_opCellDrawerCylExtend 			:BOOL:=FALSE;
//    itl_opCellDrawerCylRetract 			:BOOL:=FALSE;
//    itl_opCellDrawerCylUp 				:BOOL:=FALSE;
//    itl_opCellDrawerCylDown 			:BOOL:=FALSE;
//    itl_opTst240VACPwrEnable 			:BOOL:=FALSE;
//    itl_opCellPCWValve  				:BOOL:=FALSE;
//    itl_opAP_TIU_Skt_Air 				:BOOL:=FALSE;
//    itl_opAP_TBD						:BOOL:=FALSE;
//    itl_opAP_AirSupplySol				:BOOL:=FALSE;
//    itl_opTesterDrawerAirSupplySol	    :BOOL:=FALSE;
//    itl_opCell_24VPowerEnable			:BOOL:=FALSE;
//    itl_opCellDoorClosed				:BOOL:=FALSE;
	
END_VAR
	M_InputBackDoor();																				  
//<POC_Analog_Read>
//	IF (NOT bDebugCart AND iLevel = 3) OR (bDebugCart  AND iLevel <> 3) THEN
	aiXConverted[iLevel] := (stMLDIO.aiXAxis*8.0/32767.0)-4.0;
	aiYConverted[iLevel] := (stMLDIO.aiYAxis*8.0/32767.0)-4;
	aiY1Converted[iLevel] := (stMLDIO.aiY1Axis*8.0/32767.0)-4;
	aiZConverted[iLevel] := (stMLDIO.aiZAxis*8.0/32767.0)-4;	
	aiXConvertedRet[iLevel] := (stMLDIO.aiXAxisRet*8.0/32767.0)-4;
	aiYConvertedRet[iLevel] := (stMLDIO.aiYAxisRet*8.0/32767.0)-4;
	aiZConvertedRet[iLevel] := (stMLDIO.aiZAxisRet*8.0/32767.0)-4;
//	END_IF
//</POC_Analog_Read>

//<DrawerExtendRetract>
	stMLVIO.opCellDrawerCylExtend 	:= fbTCDrawerExtRet.P_opExtend;
	stMLVIO.opCellDrawerCylRetract 	:= fbTCDrawerExtRet.P_opRetract;
	stMLVIO.opCellDrawerCylUp 		:= fbTCDrawerUpDn.P_opExtend; 					
	stMLVIO.opCellDrawerCylDown 	:= fbTCDrawerUpDn.P_opRetract; 
//</DrawerExtendRetract>

	isLeakage:= stMLVIO.ipCellFluidLeakage1 OR stMLVIO.ipCellFluidLeakage2	;									//Used by Tst Pwr On Chk
	isGroundFault := stMLVIO.ipCellGroundFault OR ALMTC.Common.AlarmID[E_ColAlarm.ipColumnFluid_PCW_Leakage] ;	//Used by Tst Pwr On Chk
	
	IF bDebugCart = FALSE AND bDebugStation = FALSE THEN
		TBOT_TC_ACPower_Signal	:= stMLVIO.TBOT_TC_ACPower_Signal	:= stTCMLSeqParam.bTCCellACPwrOff;
	END_IF
	
	M_InterlockTII(iLevel:=iLevel);
	M_240TstPwr(iLevel:=iLevel);
	M_240APPwr(iLevel:=iLevel);
	M_Secondary24VPower(iLevel:=iLevel);
	
//inPOn :=stTCMultiLevelVIO.ipAP_PresentSensor AND stTCMultiLevelVIO.ipTesterLatchesClosed;
//delay(msec:=20000,in:=inPOn,out:=outPon);

//<ButtonLEDs>
	//stMLVIO.opDoorOpenReqLED 	:= stMLVIO.bButtons[0];
	//stMLVIO.opTCCellAbortFlowBtnLED 	:= stMLVIO.bButtons[1];
	//stMLVIO.opDrawerMaintenanceModeBtnLED 	:= stMLVIO.bButtons[2];
//</ButtonLEDs>

//<AirSupply>
	AirOnOff(); // Tester Air and AP Air
//<AirSupply>



//Do not have manual command, so we can on automatically if pass permissive.
IF bDebugCart THEN
	stMLVIO.opAPSafeToEngage	:=	(stMLVIO.ipTCDrawerCylDownRS AND stMLVIO.ipTCDrawerCylRetractRS AND NOT stMLVIO.ipTCDrawerCylExtendRS) 	//pass criteria: drawer retract: 1, drawer down: 1, drawer extend: 0
							  		//AND (stMLVIO.ipTCCellTbotSideDoorOpenCloseStatus01 AND stMLVIO.ipTCCellTbotSideDoorOpenCloseStatus02) 	//pass criteria: front door closed1&2: 1 
									//AND stMLVIO.ipTCCellDoorOpenCloseStatus 																//pass criteria: back door/ TC door closed : 1
									AND	(stMLVIO.ipTCCellTbotSideDoorLocked01 AND stMLVIO.ipTCCellTbotSideDoorLocked02)						//pass criteria: front door locked1&2: 1
									AND stMLVIO.ipTCCellDoorClosed 																			//pass criteria: back door/ TC door locked: 1
									//AND stMLVIO.opTesterDrawerAirSupplySol 																	//pass criteria: tester air 6 bar valve: 1
									AND ((NOT stMLVIO.ipTesterPresent) OR (stMLVIO.ipTesterPresent AND stMLVIO.ipTesterLatchesClosed)); 	//pass criteria: testerpresent : 0 OR tester present and tester latches closed : 1

															 	
ELSE
	stMLVIO.opAPSafeToEngage	:=	(stMLVIO.ipTCDrawerCylDownRS AND stMLVIO.ipTCDrawerCylRetractRS) 									//pass criteria: drawer retract: 1, drawer down: 1
									//AND stMLVIO.ipTCCellDoorOpenCloseStatus 															//pass criteria: back door/ TC door closed : 1
									AND stMLVIO.ipTCCellDoorClosed 																		//pass criteria: back door/ TC door locked: 1
									//AND stMLVIO.opTesterDrawerAirSupplySol  															//pass criteria: tester air 6 bar valve: 1
									AND ((NOT stMLVIO.ipTesterPresent) OR (stMLVIO.ipTesterPresent AND stMLVIO.ipTesterLatchesClosed));	//pass criteria: testerpresent : 0 OR tester present and tester latches closed : 1

	
END_IF
	
	stMLVIO.opCellPCWValve		:= (stMLVIO.ipAPPresentSensor AND NOT stMLVIO.ipTesterPresent) OR
									(stMLVIO.ipTesterPowerOn);
		
//<Output>
	IF stMLVIO.bDiagnosticMode=FALSE THEN
		stMLDIO.opAP240ACPwrEnable  			:= 		NOT	itl_opAP_240ACPwrEnable  							AND	stMLVIO.opAP240ACPwrEnable  				;//AND stMLVIO.bTstDelInt	(*&!	bTstAC	Off*)	;
		stMLDIO.opSpare_1						:=		stMLVIO.opSpare_1;
		stMLDIO.opSpare_2						:=		stMLVIO.opSpare_2;
		stMLDIO.opSpare_3						:=		stMLVIO.opSpare_3;
		stMLDIO.opDoorOpenReqLED				:= 		NOT	itl_opDoorOpenReqLED								AND	stMLVIO.opDoorOpenReqLED					;
		stMLDIO.opAlarmLED 						:= 		NOT	itl_opAlarmLED 				        				AND	stMLVIO.opAlarmLED 							;		
		stMLDIO.opTCCellAbortFlowBtnLED			:= 		NOT	itl_opTesterAPDetachReqBtnLED						AND	stMLVIO.opTCCellAbortFlowBtnLED		    	;
		stMLDIO.opDrawerMaintenanceModeBtnLED 	:= 		NOT	itl_opTesterDrawerAirOffReqBtnLED   				AND	stMLVIO.opDrawerMaintenanceModeBtnLED     	;
		stMLDIO.opAPSafeToEngage         		:= 		NOT	itl_opAP_SafeToMoveSignal           				AND	stMLVIO.opAPSafeToEngage             		;
		stMLDIO.opAPTCCReset					:= 		NOT	itl_opAP_TCCReset									AND	stMLVIO.opAPTCCReset						;	
		stMLDIO.opCellLTIMValve					:= 		NOT	itl_opCell_LTIMValve		        				AND	stMLVIO.opCellLTIMValve						;
		stMLDIO.opCellDrawerCylExtend 			:= 	    (NOT	itl_opCellDrawerCylExtend 	OR TRUE)			AND	stMLVIO.opCellDrawerCylExtend 				; //:= fbTCDrawerExtRet.P_opExtend; (* AND TBot InterLock Sen*)	
		stMLDIO.opCellDrawerCylRetract 			:= 		(NOT	itl_opCellDrawerCylRetract 	OR TRUE)			AND	stMLVIO.opCellDrawerCylRetract 				; //:= fbTCDrawerExtRet.P_opRetract ; (* OR (NOT fbTCDrawerIn.P_opRetract AND TBot InterLock Sen) *)	
		stMLDIO.opCellDrawerCylUp 				:= 		(NOT	itl_opCellDrawerCylUp 		OR TRUE)			AND stMLVIO.opCellDrawerCylUp 					; //:= fbTCDrawerUpDn.P_opExtend; 		
		stMLDIO.opCellDrawerCylDown 			:= 		(NOT	itl_opCellDrawerCylDown 	OR TRUE)			AND	stMLVIO.opCellDrawerCylDown 				; //:= fbTCDrawerUpDn.P_opRetract; 
		stMLDIO.opTst240VACPwrEnable 			:= 		NOT	itl_opTst240VACPwrEnable 							AND	stMLVIO.opTst240VACPwrEnable 				;
		stMLDIO.opSpare_9						:=		stMLVIO.opSpare_9;
		stMLDIO.opSpare_10						:=		stMLVIO.opSpare_10;
		stMLDIO.opCellPCWValve  				:= 		NOT	itl_opCellPCWValve  			    				AND	stMLVIO.opCellPCWValve  					;	//AND stMLVIO.bTstDelInt	;
		stMLDIO.opTIUSktAirSol_1 				:= 		NOT	itl_opTIUSktAirSol_1 								AND stMLVIO.opTIUSktAirSol_1 					;
		stMLDIO.opTIUSktAirSol_2				:= 		NOT	itl_opTIUSktAirSol_2								AND stMLVIO.opTIUSktAirSol_2					;	
		stMLDIO.opAPAirSupplySol				:= 		NOT	itl_opAP_AirSupplySol 								AND stMLVIO.opAPAirSupplySol					;
		stMLDIO.opTesterDrawerAirSupplySol		:= 		NOT	itl_opTesterDrawerAirSupplySol	    				AND stMLVIO.opTesterDrawerAirSupplySol	    	;
		stMLDIO.opCell24VPowerEnable			:= 		NOT	itl_opCell_24VPowerEnable							AND	stMLVIO.opCell24VPowerEnable				;			    //AND stMLVIO.bTstDelInt  ;
		stMLDIO.opCellDoorClosed				:= 	   (NOT itl_opCellDoorClosed OR TRUE)						AND stMLVIO.opCellDoorClosed					;
		stMLDIO.opCellTBOtSideDoorClosed1		:= 		stMLVIO.opCellTBOtSideDoorClosed1					;
		stMLDIO.opCellTBOtSideDoorClosed2		:= 		stMLVIO.opCellTBOtSideDoorClosed2					;
		
	ELSE
		stTCColVIO:=  fbTCColumn.P_stTCColumnVIO;
		IF 	M_IsEAPError()> 0 OR 
			( bDebugCart AND 	(stMLDIO.ipTCCellTbotSideDoorOpenCloseStatus01 OR stMLDIO.ipTCCellTbotSideDoorLocked01) OR (stMLDIO.ipTCCellTbotSideDoorOpenCloseStatus02 OR stMLDIO.ipTCCellTbotSideDoorLocked02)) OR  
			( stMLVIO.ipAPPresentSensor  AND NOT (stMLVIO.ipHandlerSafeToEnterHwr AND stMLVIO.ipHandlerSafeToEnterPLC) AND NOT stMLVIO.ipAPReady ) //OR 
		(*(stMLVIO.ipCellFluidLeakage1 OR stMLVIO.ipCellFluidLeakage1 OR stTCColVIO.ipColumnFluid_PCW_Leakage )*) THEN		
			stMLDIO.opCellDrawerCylExtend		:= 		(NOT	itl_opCellDrawerCylExtend 	OR TRUE		)AND	stMLVIO.opCellDrawerCylExtend 				; 
			stMLDIO.opCellDrawerCylRetract		:= 		(NOT	itl_opCellDrawerCylRetract 	OR TRUE		)AND	stMLVIO.opCellDrawerCylRetract 				; 	
			//stMLDIO.opCellDrawerCylUp			:= 		(NOT	itl_opCellDrawerCylUp 		OR TRUE		)AND 	stMLVIO.opCellDrawerCylUp 					; 
			//stMLDIO.opCellDrawerCylDown			:= 		(NOT	itl_opCellDrawerCylDown 	OR TRUE		)AND	stMLVIO.opCellDrawerCylDown 			    ; 
		END_IF                                                                                                                                                    		
		(*
		//<DrawerExtendRetract>
			stMLVIO.opCellDrawerCylExtend 	:= fbTCDrawerExtRet.P_opExtend		:= 	stMLDIO.opCellDrawerCylExtend 	;
			stMLVIO.opCellDrawerCylRetract 	:= fbTCDrawerExtRet.P_opRetract     :=  stMLDIO.opCellDrawerCylRetract 	;
			stMLVIO.opCellDrawerCylUp 		:= fbTCDrawerUpDn.P_opExtend		:= 	stMLDIO.opCellDrawerCylUp 		;		
			stMLVIO.opCellDrawerCylDown 	:= fbTCDrawerUpDn.P_opRetract       :=  stMLDIO.opCellDrawerCylDown 	;
		//</DrawerExtendRetract>
		*)
	END_IF
//</Output>
END_METHOD

METHOD M_IsEAPError : INT
VAR_INPUT
END_VAR

VAR_OUTPUT
	sMsg					: STRING;
END_VAR
// Receive drawer not safe to move from TBOT
IF stTCMLSeqParam.bTCDwrSafeToMoveEAP = FALSE THEN 
	sMsg									:= 'TBot EAP not safe to move!';;
	M_IsEAPError							:= E_AlarmID.TBotEAPNotSafeToMoveError; //25;
// Receive anti-collision signal from TBOT
ELSIF (NOT stTCMLSeqParam.bTBotAntiCollisionTriggered) THEN
	sMsg									:= 'TBotAntiCollisionTriggered Error';
	M_IsEAPError							:= E_AlarmID.TBotEAPAntiCollisionTriggered;//26;
END_IF
END_METHOD

METHOD M_nCmptInOut : UDINT
VAR_INPUT
	bExtend						: BOOL;
END_VAR

VAR
END_VAR

VAR_IN_OUT
	sErrorMsg 					: STRING;
END_VAR
IF bExtend THEN
	iLibrySts[1]					:= inTCDrawerExtRet.M_nExtend(bExecute:= TRUE);
ELSE
	iLibrySts[1]					:= inTCDrawerExtRet.M_nRetract(bExecute:= TRUE);
END_IF

IF iLibrySts[1] = 10 THEN
	inTCDrawerExtRet.M_nOff();
	M_nCmptInOut					:= 10;
ELSIF inTCDrawerExtRet.P_bError THEN
	sErrorMsg						:= CONCAT(sMessage,fbTCDrawerExtRet.P_sMessage);
	stMLVIO.iAlarmCode				:= inTCDrawerExtRet.P_nErrorID;
	M_nCmptInOut					:= 99;
END_IF
END_METHOD

METHOD M_nCmptUpDown : UDINT
VAR_INPUT
	bExtend					: BOOL;
END_VAR

VAR
END_VAR

VAR_IN_OUT
	sErrorMsg				: STRING;
END_VAR
	
	
IF bExtend THEN
	iLibrySts[1]					:= inTCDrawerUpDn.M_nExtend(bExecute:= TRUE);
ELSE
	iLibrySts[1]					:= inTCDrawerUpDn.M_nRetract(bExecute:= TRUE);
END_IF

IF iLibrySts[1] = 10 THEN
	inTCDrawerUpDn.M_nOff();
	M_nCmptUpDown					:= 10;
ELSIF inTCDrawerUpDn.P_bError THEN
	sErrorMsg						:= CONCAT(sMessage,fbTCDrawerUpDn.P_sMessage);
	stMLVIO.iAlarmCode				:= inTCDrawerUpDn.P_nErrorID;
	M_nCmptUpDown					:= 99;
END_IF
END_METHOD

METHOD M_nCyclic : UDINT
VAR_INPUT
	iLevel:INT;
END_VAR


VAR
	//stTCM: INT;
	stGblParam: INT;
	varTest:bool;
END_VAR
//M_nCompCylinder(bExtend:=TRUE, fbTCDrawerUp, sMsg);
//M_IOMapping();

M_IOMapping(iLevel:=iLevel);

rtError(CLK:=_bError, Q=> );
btest:=TRUE;

	fbTCDrawerExtRet.M_nReset(bExecute:=_bReset OR rtError.Q );
	fbTCDrawerUpDn.M_nReset(bExecute:=_bReset OR rtError.Q );
		
IF _bReset OR bStepDone OR rtError.Q THEN
	inTCDrawerExtRet.M_nOff();
	inTCDrawerUpDn.M_nOff();
	
	//sensor

	FOR nI:=1 TO 20 DO 
		iLibrySts[1] := 0;
	END_FOR
	
	bStepDone:=FALSE; 
END_IF

inTCDrawerExtRet.P_SensorDelay:= tDwrCylExtRetSensorDelay;	//FB_M_nCyclic_tSensorDelay  ;  //T#12S; 
inTCDrawerExtRet.P_Timeout:= 	tDwrCylExtRetTimeOut;	//FB_M_nCyclic_tSensorTimeOut; //T#30S;;    

inTCDrawerUpDn.P_SensorDelay:= tDwrCylUpDownSensorDelay; //FB_M_nCyclic_tSensorDelay;
inTCDrawerUpDn.P_Timeout:= tDwrCylUpDownTimeOut;//FB_M_nCyclic_tSensorTimeOut;

(*IF stTCSeqParam.bInitComplt THEN //temp...This portion will be done by Initialise sequence
END_IF*)
	
IF _bReset THEN
	IF stTCMLSeqParam.bInitialise THEN
		iSysRsetSeqStep:=0;
	ELSE
		iSeqStep:=0;
	END_IF
	iStkSeqCase:=0;
	bStepDone:=FALSE;
	sMessage:='';
	_bError:=FALSE;
	_nErrorID:=0;
ELSIF bErrClear THEN
	_bError:=FALSE;
	_nErrorID:=0;
	bErrClear:=FALSE;
END_IF

bPause:=_bReset OR _bError OR bErrClear;
//M_StkSingStackUp state
IF _bError THEN
	iStkSingStackUp:=99;
ELSIF _bReset THEN
	iStkSingStackUp:=0;
ELSIF iStkSeqCase=E_SeqSts.eDone THEN
	iStkSingStackUp:=10;
ELSIF NOT bPause THEN
	iStkSingStackUp:=3;
END_IF

inTCDrawerExtRet.P_nExtendAlarmID:=E_AlarmID.DrawerExtendError;
inTCDrawerExtRet.P_nRetractAlarmID:=E_AlarmID.DrawerRetractError;
inTCDrawerUpDn	 .P_nExtendAlarmID:=E_AlarmID.DrawerUpError;
inTCDrawerUpDn	 .P_nRetractAlarmID:=E_AlarmID.DrawerDownError;

//<IN_OUT>
	IF stMLVIO.ipTCDrawerCylRetractRS AND NOT stMLVIO.ipTCDrawerCylExtendRS THEN
		stMLVIO.bTIUInOutStatusFlag:= FALSE;
	ELSE
		stMLVIO.bTIUInOutStatusFlag:= TRUE;
	END_IF
//</IN_OUT>
//<UP_DOWN>
	IF stMLVIO.ipTCDrawerCylDownRS AND NOT stMLVIO.ipTCDrawerCylUpRS THEN
		stMLVIO.bTIUUpDownStatusFlag:= FALSE;
	ELSE
		stMLVIO.bTIUUpDownStatusFlag:= TRUE;
	END_IF
//</UP_DOWN>
//<DCCell_DoorStatus>
	IF bDebugCart THEN
	(*
		stMLVIO.opCellFrontDoorClosedStatus		:= 	stMLVIO.opCellFrontDoorClosed1 AND stMLVIO.opCellFrontDoorClosed2;
		stMLVIO.ipTCCellFrontDoorLockedStatus	:= 	stMLVIO.opCellFrontDoorClosed1 AND stMLVIO.opCellFrontDoorClosed2; //stMLVIO.ipTCCellFrontDoorOpenCloseStatus1 AND stMLVIO.ipTCCellFrontDoorOpenCloseStatus2;
	*)
	//(*
		stMLVIO.bCellFrontDoorLockedStatus	:= 	stMLVIO.opCellTBOtSideDoorClosed1 AND stMLVIO.opCellTBOtSideDoorClosed2;
		stMLVIO.bCellFrontDoorClosedStatus 	:= 	stMLVIO.ipTCCellTbotSideDoorOpenCloseStatus01 AND stMLVIO.ipTCCellTbotSideDoorOpenCloseStatus02;
	//*)
		
	END_IF
//</DCCell_DoorStatus>


stMLVIO.opAlarmLED:= stMLVIO.TIIAlarmLED OR _bError OR stMLVIO.isSysError;
END_METHOD

METHOD M_nDPSPowerOnOff : INT
VAR_INPUT
END_VAR
VAR
END_VAR
M_nDPSPowerOnOff:=iStkSingStackUp;

IF bPause THEN
	RETURN;

ELSIF itl_opTst240VACPwrEnable AND stTCMLSeqParam.bDSPPowerOn THEN  
	M_nDPSPowerOnOff						:= 20;		
	RETURN;
ELSIF itl_opAP_240ACPwrEnable AND stTCMLSeqParam.bAP240ACPowerOn THEN
	M_nDPSPowerOnOff						:= 20;
	RETURN;
END_IF

IF iSeqStep>0 THEN
	;//Do nothing;
ELSIF stTCMLSeqParam.bDSPPowerOff OR
	  stTCMLSeqParam.bDSPPowerOn OR
	  stTCMLSeqParam.bDSPPowerAuto 
	  THEN
	arrSeqStep[0]:=E_SeqSts.eInit;					//Init
	arrSeqStep[1]:=E_SeqSts.eSanityCheckForDPSPwr;	//Sanity check
	arrSeqStep[2]:=E_SeqSts.eDPSPwrOnOff;			//DPSPowerOnOff
	arrSeqStep[3]:=E_SeqSts.eDone;					//Done
	
ELSIF stTCMLSeqParam.bAP240ACPowerOff OR
	  stTCMLSeqParam.bAP240ACPowerOn OR
	  stTCMLSeqParam.bAP240ACPowerAuto 
	  THEN
	arrSeqStep[0]:=E_SeqSts.eInit;						//Init
	arrSeqStep[1]:=E_SeqSts.eSanityCheckForAPPwr;		//Sanity check
	arrSeqStep[2]:=E_SeqSts.eAP240ACPwrOnOff;			//AP240ACPowerOnOff
	arrSeqStep[3]:=E_SeqSts.eDone;						//Done
	
END_IF

//Sequence start
iStkSeqCase:=arrSeqStep[iSeqStep];

// State machine
CASE iStkSeqCase OF
	E_SeqSts.eInit: //Init
		//TDelay(IN:=FALSE);
		sMessage:='Start Executing';
		bStepDone:=TRUE;
		
	E_SeqSts.eSanityCheckForDPSPwr: 			//Sanity check DPS
		sMessage:='CheckTeir2IIAlarm';
		
		tDPSDelayToComplete(IN:=FALSE);
		tDPSDelayToAutoComplete(IN:=FALSE);
		bStepDone:=TRUE;
	
	E_SeqSts.eSanityCheckForAPPwr: 				//Sanity check AP
		sMessage:='CheckTeir2IIAlarm';
		
		tAPACPwrDelayToComplete(IN:=FALSE);
		tAPACPwrDelayToAutoComplete(IN:=FALSE);
		bStepDone:=TRUE;	
		
		
	E_SeqSts.eDPSPwrOnOff:											// DSPPowerOnOff
		tDPSDelayToComplete(IN:=TRUE, PT:=T#2S); 				// origin T#10s
		IF tDPSDelayToComplete.Q THEN
			IF stTCMLSeqParam.bDSPPowerOff THEN 				(*0=Off, 1=On, 2=Auto(Off->On) *)
				stMLVIO.bDPSPowerOnOff:=FALSE;//TRUE;
				tDPSDelayToAutoComplete(IN:=TRUE, PT:=T#0S);
				sMessage:='DSPPowerOff';
			ELSIF stTCMLSeqParam.bDSPPowerON THEN
				stMLVIO.bDPSPowerOnOff:=TRUE;//FALSE;
				tDPSDelayToAutoComplete(IN:=TRUE, PT:=T#0S);
				sMessage:='DSPPowerOn';
			ELSIF  stTCMLSeqParam.bDSPPowerAuto THEN
				stMLVIO.bDPSPowerOnOff:=FALSE;//TRUE;
				sMessage:='DSPPowerOff';
				tDPSDelayToAutoComplete(IN:=TRUE, PT:=T#2S);	// origin T#10s
				IF tDPSDelayToAutoComplete.Q THEN
					stMLVIO.bDPSPowerOnOff:=TRUE;//FALSE;	
					sMessage:='DSPPowerOn';
				END_IF
			END_IF
		END_IF
		
		IF tDPSDelayToComplete.Q AND tDPSDelayToAutoComplete.Q THEN
			tDPSDelayToComplete(IN:=FALSE);
			tDPSDelayToAutoComplete(IN:=FALSE);
			bStepDone:=TRUE;
		END_IF
	
	E_SeqSts.eAP240ACPwrOnOff:										// AP240ACPowerOnOff
		tAPACPwrDelayToComplete(IN:=TRUE, PT:=T#2S); 			// origin T#10s
		IF tAPACPwrDelayToComplete.Q THEN
			IF stTCMLSeqParam.bAP240ACPowerOff THEN 			(*0=Off, 1=On, 2=Auto(Off->On) *)
				stMLVIO.bAP240ACPowerOnOff		:=FALSE;//TRUE;
				tAPACPwrDelayToAutoComplete(IN:= TRUE, PT:=T#0S);
				sMessage:='AP240AC PowerOff';
			ELSIF stTCMLSeqParam.bAP240ACPowerOn THEN
				stMLVIO.bAP240ACPowerOnOff		:= TRUE;//FALSE;
				tAPACPwrDelayToAutoComplete(IN:=TRUE, PT:=T#0S);
				sMessage:='AP240AC PowerOn';
			ELSIF  stTCMLSeqParam.bAP240ACPowerAuto THEN
				stMLVIO.bAP240ACPowerOnOff		:= FALSE;//TRUE;
				sMessage:='AP240AC PowerOff';
				tAPACPwrDelayToAutoComplete(IN:=TRUE, PT:=T#2S); // origin T#10s
				IF tAPACPwrDelayToAutoComplete.Q THEN
					stMLVIO.bAP240ACPowerOnOff		:= TRUE;//FALSE;
					sMessage:='AP240AC PowerOn';
				END_IF
			END_IF
		END_IF
			
		IF tAPACPwrDelayToComplete.Q AND tAPACPwrDelayToAutoComplete.Q THEN
			tAPACPwrDelayToComplete(IN:=FALSE);
			tAPACPwrDelayToAutoComplete(IN:=FALSE);
			bStepDone:=TRUE;
		END_IF
	
	E_SeqSts.eDone:	// Done
		sMessage:='Done';
		M_nDPSPowerOnOff:=10;
		
END_CASE	

IF (bStep OR bBypassSingleMove OR iStkSeqCase<=E_SeqSts.eSanityCheck) AND iStkSeqCase<E_SeqSts.eDone AND bStepDone THEN
	iSeqStep:=iSeqStep+1;
END_IF

rtStep(CLK:=bStep AND NOT bBypassSingleMove, Q=>bStep );
END_METHOD

METHOD M_Pwr : bool
VAR_INPUT
	e:BOOL;
END_VAR

	//stMLVIO.opAP240ACPwrEnable:=
	//stMLVIO.opCell24VPowerEnable:=
	//stMLVIO.opTst240VACPwrEnable:=
	//stMLVIO.opCellPCWValve:=
	//stMLVIO.bEnableSKTAirSupOnInit:=
	//stMLVIO.bEnableAPPwrSupOnInit:=
	stMLVIO.bEnableAPAirSupOnInit:=
	//stMLVIO.bEnableTstPwrSupOnInit:=
	stMLVIO.bEnableDwrAirSupOnInit:=
	FunONOFF:= 
	e;
END_METHOD

METHOD M_RemoteSecondary24VPowerOnOff : INT
VAR_INPUT
END_VAR
IF bPause THEN
	RETURN;
	
ELSIF itl_opCell_24VPowerEnable OR stMLVIO.isSysError THEN
	M_RemoteSecondary24VPowerOnOff				:= 20;		
	RETURN;
END_IF

IF stTCMLSeqParam.bSecondary24VPowerOff THEN
	stMLVIO.bSecondary24VPowerOnOff				:= FALSE;
	M_RemoteSecondary24VPowerOnOff				:= 10;
	
ELSIF stTCMLSeqParam.bSecondary24VPowerOn THEN
	stMLVIO.bSecondary24VPowerOnOff				:= TRUE;
	M_RemoteSecondary24VPowerOnOff				:= 10;
END_IF
END_METHOD

METHOD M_Secondary24VPower : UDINT
VAR_INPUT
	iLevel:INT;
END_VAR
VAR
	Permissive_opCell24VPowerEnable			: WORD;
	Shutdown_opCell24VPowerEnable			: WORD;
END_VAR
FC_BitToWord(
	BOOL_00		:= TRUE, 
	BOOL_01		:= TRUE, 
	BOOL_02		:= TRUE, 
	BOOL_03		:= TRUE, 
	BOOL_04		:= TRUE, 
	BOOL_05		:= TRUE, 
	BOOL_06		:= TRUE, 
	BOOL_07		:= TRUE, 
	BOOL_08		:= TRUE, 
	BOOL_09		:= TRUE, 
	BOOL_10		:= TRUE, 
	BOOL_11		:= TRUE, 
	BOOL_12		:= TRUE, 
	BOOL_13		:= TRUE, 
	BOOL_14		:= TRUE, 
	BOOL_15		:= TRUE, 
	Output_Word		=> Permissive_opCell24VPowerEnable);
	
FC_BitToWord(
	BOOL_00		:= FALSE, 
	BOOL_01		:= FALSE, 
	BOOL_02		:= FALSE, 
	BOOL_03		:= FALSE, 
	BOOL_04		:= FALSE, 
	BOOL_05		:= FALSE, 
	BOOL_06		:= FALSE, 
	BOOL_07		:= FALSE, 
	BOOL_08		:= FALSE, 
	BOOL_09		:= FALSE, 
	BOOL_10		:= FALSE, 
	BOOL_11		:= FALSE, 
	BOOL_12		:= FALSE, 
	BOOL_13		:= FALSE, 
	BOOL_14		:= FALSE, 
	BOOL_15		:= FALSE, 
	Output_Word		=> Shutdown_opCell24VPowerEnable);
	

Precondition_opCell24VPowerEnable		:=  (NOT itl_opCell_24VPowerEnable) AND 
											stMLVIO.bSecondary24VPowerOnOff;

Reset_opCell24VPowerEnable(CLK:= Precondition_opCell24VPowerEnable);
			
DUT_opCell24VPowerEnable.AutInp			:= Precondition_opCell24VPowerEnable;
DUT_TC_AP240ACPower.Reset		:= Reset_opCell24VPowerEnable.Q;						
	
FB_opCell24VPowerEnable(
	Sec_P:= Sec_P, 
	ID:= 'Cell 24V Secondary Power', 
	Simulate:= DUT_opCell24VPowerEnable.Simulate, 
	Permissive:= Permissive_opCell24VPowerEnable,  //check before execute
	ShutDown:= Shutdown_opCell24VPowerEnable,  //keep checking this condition 
	AutoInp:= DUT_opCell24VPowerEnable.AutInp, 
	Command:= DUT_opCell24VPowerEnable.CMD, //1: Retract, 2: Extend, 4: Auto
	IExtend:= stMLVIO.opCell24VPowerEnable, 
	IRetract:= (NOT stMLVIO.opCell24VPowerEnable), 
	Travel_Time:= DUT_opCell24VPowerEnable.Travel_Time, //detect input after output trigger
	SetOutput_Pulse:= FALSE,  //output rising edge
	FailedHoldLast:= FALSE,  //remain state after failed. 1: Remain, 0: FALSE
	OExtend=> stMLVIO.opCell24VPowerEnable,  //map to output variable
	ORetract=> , 
	DUT:= DUT_opCell24VPowerEnable);
END_METHOD

METHOD M_SeqAlmRset : UDINT
VAR_INPUT
	subMod:DINT;
	almID:DINT;
	isRsetAll:BOOL;
END_VAR
VAR
	i:UINT;
END_VAR
IF isRsetAll THEN
	FOR i:=1 TO NO_OF_ALARM_TAG DO
		ALMTC.Level[subMod].AlarmID[i] := FALSE;
	END_FOR
ELSE
	ALMTC.Level[subMod].AlarmID[almID] := FALSE;
END_IF
END_METHOD

METHOD M_SequenceCommand : INT
VAR_INPUT
	iLevel		: UINT;
END_VAR
VAR
	stColVIO					: ST_TCColumn_VIO;
	isError						: BOOL;
	sDebugLog					: STRING; 
	lrPosition					: LREAL;
	i							: INT; //for loop
	addEvntOk					: BOOL;
	iTIUStatus					: INT;
END_VAR
M_SequenceCommand										:= iStkSingStackUp;

IF (bPause) THEN
	RETURN;
END_IF

///////////////////////////////////////////////////////////////////////////////////////////////////////////////////////////////////////////////////////////////////////////////
//	State Assignment
///////////////////////////////////////////////////////////////////////////////////////////////////////////////////////////////////////////////////////////////////////////////

IF iSeqStep > 0 THEN
	;//Do nothing;
ELSIF stTCMLSeqParam.bDrawerUp THEN
	iStkSeqCase												:= 0;
	arrSeqStep[0]											:= E_SeqSts.eInit;
	arrSeqStep[1]											:= E_SeqSts.eDrawerUpDownSanityCheck;
	arrSeqStep[2]											:= E_SeqSts.eMoveDrawerUp;
	arrSeqStep[3]											:= E_SeqSts.eDone;		
	
ELSIF stTCMLSeqParam.bDrawerDown THEN
	iStkSeqCase 											:= 0; 						
	arrSeqStep[0]											:= E_SeqSts.eInit;			
	arrSeqStep[1]											:= E_SeqSts.eDrawerUpDownSanityCheck;	
	arrSeqStep[2]											:= E_SeqSts.eMoveDrawerDown;
	arrSeqStep[3]											:= E_SeqSts.eDone;	
	
ELSIF stTCMLSeqParam.bCancel THEN
	iStkSeqCase := 0;
	arrSeqStep[0]											:= E_SeqSts.eInit;
	arrSeqStep[1]											:= E_SeqSts.eDrawerUpDownInOutSanityCheck;
	arrSeqStep[2]											:= E_SeqSts.eTBotEAPSanityCheck;
	arrSeqStep[3]											:= E_SeqSts.eMoveDrawerUp;
	arrSeqStep[4]											:= E_SeqSts.eTBotEAPSanityCheck;
	arrSeqStep[5]											:= E_SeqSts.eMoveDrawerIn;
	arrSeqStep[6]											:= E_SeqSts.eMoveDrawerDown;
	arrSeqStep[7]											:= E_SeqSts.eDone;
	
ELSIF stTCMLSeqParam.bShuttleMoveOut OR stTCMLSeqParam.bTBotbShuttleMoveOutReq THEN
	arrSeqStep[0]											:= E_SeqSts.eInit;
	arrSeqStep[1]											:= E_SeqSts.eDrawerUpDownInOutSanityCheck;
	arrSeqStep[2]											:= E_SeqSts.eTBotEAPSanityCheck;
	arrSeqStep[3]											:= E_SeqSts.eMoveDrawerUp;
	arrSeqStep[4]											:= E_SeqSts.eTBotEAPSanityCheck;
	arrSeqStep[5]											:= E_SeqSts.eMoveDrawerOut;
	arrSeqStep[6]											:= E_SeqSts.eDone;

ELSIF stTCMLSeqParam.bDrawerUpBefFrtDoorOpen THEN
	arrSeqStep[0]											:= E_SeqSts.eInit;
	arrSeqStep[1]											:= E_SeqSts.eFrontDoorOpenConditionCheck;
	arrSeqStep[2]											:= E_SeqSts.eDrawerUpDownSanityCheck;
	arrSeqStep[3]											:= E_SeqSts.eMoveDrawerUp;
	arrSeqStep[4]											:= E_SeqSts.eMoveDrawerOut; //eOnDrawerOutputOnly
	arrSeqStep[5]											:= E_SeqSts.eTurnOffAPAirValve;
	arrSeqStep[6]											:= E_SeqSts.eTurnOffTesterAirValve;
	arrSeqStep[7]											:= E_SeqSts.eUnlockFrontDoor;
	arrSeqStep[8]											:= E_SeqSts.eDone;

ELSIF stTCMLSeqParam.bShuttleMoveIn OR stTCMLSeqParam.bDoorRecovery OR stTCMLSeqParam.bTBotbShuttleMoveInReq THEN
	arrSeqStep[0]											:= E_SeqSts.eInit;
	arrSeqStep[1]											:= E_SeqSts.eDrawerUpDownInOutSanityCheck;
	arrSeqStep[2]											:= E_SeqSts.eChkTIUPosition;
	arrSeqStep[3]											:= E_SeqSts.eTBotEAPSanityCheck;
	arrSeqStep[4]											:= E_SeqSts.eMoveDrawerUp;
	arrSeqStep[5]											:= E_SeqSts.eTBotEAPSanityCheck;
	arrSeqStep[6]											:= E_SeqSts.eMoveDrawerIn;
	arrSeqStep[7]											:= E_SeqSts.eTurnOnTesterAirValve;
	arrSeqStep[8]											:= E_SeqSts.eMoveDrawerDown;
	arrSeqStep[9]											:= E_SeqSts.eTurnOnAPAirValve;
	arrSeqStep[10]											:= E_SeqSts.eDone;
END_IF

///////////////////////////////////////////////////////////////////////////////////////////////////////////////////////////////////////////////////////////////////////////////
//	Current sequence case
///////////////////////////////////////////////////////////////////////////////////////////////////////////////////////////////////////////////////////////////////////////////

iStkSeqCase													:= arrSeqStep[iSeqStep];

///////////////////////////////////////////////////////////////////////////////////////////////////////////////////////////////////////////////////////////////////////////////
//	State machine
///////////////////////////////////////////////////////////////////////////////////////////////////////////////////////////////////////////////////////////////////////////////

CASE iStkSeqCase OF
	
///////////////////////////////////////////////////////////////////////////////////////////////////////////////////////////////////////////////////////////////////////////////
//	State: Front door open check, if drawer up signal direct skip to turn off air valves and unlock door.
///////////////////////////////////////////////////////////////////////////////////////////////////////////////////////////////////////////////////////////////////////////////	
	E_SeqSts.eFrontDoorOpenConditionCheck:
		sMessage											:= ' Drawer Up Condition Checking';
		IF stMLVIO.ipTCDrawerCylUpRS THEN
			iSeqStep										:= 5; 	//jump to turn off air valves
		ELSE
			bStepDone										:= TRUE; 
		END_IF
		
///////////////////////////////////////////////////////////////////////////////////////////////////////////////////////////////////////////////////////////////////////////////
//	State: Front door open check, if drawer up signal direct skip to unlock front door.
///////////////////////////////////////////////////////////////////////////////////////////////////////////////////////////////////////////////////////////////////////////////			
	E_SeqSts.eUnlockFrontDoor:
		stMLVIO.opCellTBOtSideDoorClosed1					:= FALSE;
		stMLVIO.opCellTBOtSideDoorClosed2					:= FALSE;
		bStepDone											:= TRUE;
		
///////////////////////////////////////////////////////////////////////////////////////////////////////////////////////////////////////////////////////////////////////////////
//	State: Initiate or Stay IDLE 
///////////////////////////////////////////////////////////////////////////////////////////////////////////////////////////////////////////////////////////////////////////////	
	E_SeqSts.eInit:
		sMessage											:= ' Start Executing';
		
		IF stTCMLSeqParam.bInitialise THEN
			;
		END_IF
		bStepDone											:= TRUE;
		
///////////////////////////////////////////////////////////////////////////////////////////////////////////////////////////////////////////////////////////////////////////////
//	State: Sanity check for different sequences
///////////////////////////////////////////////////////////////////////////////////////////////////////////////////////////////////////////////////////////////////////////////			
	E_SeqSts.eDrawerUpDownSanityCheck:
		sMessage											:= ' Drawer UpDown Sanity Check';
		_nErrorID											:= INT_TO_UDINT(M_APSanityCheck(
																				stMultiLevelVIO		:= stMLVIO,
																				sMsg				:= sMessage
																			));
		// back door lock signal alarm																	
		IF (NOT stMLVIO.ipTCCellDoorOpenCloseStatus) THEN
			sMessage									:= 'Door Closed Signal not Detected';
			_nErrorID									:= E_AlarmID.DoorCloseSignalNotDetected;//31;
		ELSIF (NOT stMLVIO.ipTCCellDoorClosed) THEN
			sMessage									:= 'Door Locked Signal not Detected';
			_nErrorID									:= E_TIIAlarm.ipTCCellDoorClosed;//12;
		END_IF
		
		// Front door lock signal alarm
		IF bDebugCart THEN 
			IF (NOT stMLVIO.ipTCCellTbotSideDoorOpenCloseStatus01) THEN
				sMessage									:= 'Front Door Closed_1 Signal not Detected';
				_nErrorID									:= E_AlarmID.TBotSideDoorCloseSignalNotDetected;//33;
			ELSIF (NOT stMLVIO.ipTCCellTbotSideDoorOpenCloseStatus02) THEN
				sMessage									:= 'Front Door Closed_2 Signal not Detected';
				_nErrorID									:= E_AlarmID.TBotSideDoorCloseSignalNotDetected;//33;
			ELSIF (NOT stMLVIO.ipTCCellTbotSideDoorLocked01) THEN
				sMessage									:= 'Front Door Lock_1 Signal not Detected';
				_nErrorID									:= E_TIIAlarm.FrontDoorLockSignalNotDetected;//34;
			ELSIF (NOT stMLVIO.ipTCCellTbotSideDoorLocked02) THEN
				sMessage									:= 'Front Door Lock_2 Signal not Detected';
				_nErrorID									:= E_TIIAlarm.FrontDoorLockSignalNotDetected;//34;
			END_IF
		END_IF 		
			
		IF _nErrorID = 0 THEN
			bStepDone										:= TRUE;
		END_IF
		
	E_SeqSts.eDrawerUpDownInOutSanityCheck: //Sanity sheck for 
		sMessage											:= ' Drawer UpDownInOut Sanity Check';
		//stColVIO											:= fbTCColumn.P_stTCColumnVIO;
		_nErrorID											:= INT_TO_UDINT(M_APSanityCheck(
																				stMultiLevelVIO		:= stMLVIO, 
																				//stColVIO			:= stColVIO, 
																				sMsg				:= sMessage
																			));
		
		// back door close signal alarm																	
		IF (NOT stMLVIO.ipTCCellDoorOpenCloseStatus) THEN
			sMessage									:= 'Door Closed Signal not Detected';
			_nErrorID									:= E_AlarmID.DoorCloseSignalNotDetected;//31;
			
		// back door lock signal alarm
		ELSIF (NOT stMLVIO.ipTCCellDoorClosed) THEN
			sMessage									:= 'Door Locked Signal not Detected';
			_nErrorID									:= E_TIIAlarm.ipTCCellDoorClosed;//12;
		END_IF	
		
		
		// drawer up signal alarm
		IF ALMTC.Level[iLevel].AlarmID[E_TIIAlarm.ipTCDrawerUpSignal] THEN
			sMessage									:= 'Drawer Up Signal not detected';
			_nErrorID									:= E_TIIAlarm.ipTCDrawerUpSignal;
			
		// drawer extend alarm
		ELSIF ALMTC.Level[iLevel].AlarmID[E_TIIAlarm.ipTCDrawerExtendSignal] THEN
			sMessage									:= 'Drawer Extend Signal not detected';
			_nErrorID									:= E_TIIAlarm.ipTCDrawerExtendSignal;
		
		// drawer retract alarm
		ELSIF ALMTC.Level[iLevel].AlarmID[E_TIIAlarm.ipTCDrawerRetractSignal] THEN
			sMessage									:= 'Drawer Retract Signal not detected';
			_nErrorID									:= E_TIIAlarm.ipTCDrawerRetractSignal;
			
		// tester latch alarm	
		ELSIF ALMTC.Level[iLevel].AlarmID[E_TIIAlarm.ipTesterLatchesClosed] THEN
			sMessage									:= 'Tester Latches Signal not detected';
			_nErrorID									:= E_TIIAlarm.ipTesterLatchesClosed;
		END_IF					

									
		IF _nErrorID = 0 THEN
			bStepDone										:= TRUE;
		END_IF
		
///////////////////////////////////////////////////////////////////////////////////////////////////////////////////////////////////////////////////////////////////////////////
//	State: Check TIU position, alarm if both signal detected // donno using or not.
///////////////////////////////////////////////////////////////////////////////////////////////////////////////////////////////////////////////////////////////////////////////			
	eChkTIUPosition:
		iTIUStatus											:= M_GetTIUStatus(
																	b3:= stMLVIO.ipTCDrawerCylUpRS,			//UP
																	b2:= stMLVIO.ipTCDrawerCylDownRS,		//DOWN
																	b1:= stMLVIO.ipTCDrawerCylExtendRS,		//EXTEND
																	b0:= stMLVIO.ipTCDrawerCylRetractRS		//RETRACT
																);
		CASE iTIUStatus OF 
			0: (*No drawer position feedback signal*)	
				bStepDone									:= TRUE;
			1: (*Drawer is retracted but no Up or Down signal*)		
				iSeqStep									:= 6; 
			2: (*Drawer is extended but no Up or Down signal*)	
				bStepDone									:= TRUE;
			3: (*Error - Receive drawer extended and retracted signal*)		
				_nErrorID									:= E_AlarmID.BothTIUUpDownSignalDetected; 
				sMessage									:= 'Both Reed Switchs of Cylinder are Detected';
			4: (*Drawer is Down but no retracted or extended signal*)	
				bStepDone									:= TRUE;
			5: (*Drawer is retracted and Down*)		
				iSeqStep									:= 6; 
			6: (*Drawer is extended and Down*)	
				bStepDone									:= TRUE;
			7: (*Error - Receive drawer is down, extended and retracted signal*)		
				_nErrorID									:= E_AlarmID.BothTIUUpDownSignalDetected; 
				sMessage									:= 'Both Reed Switchs OF Cylinder are Detected';
			8: (*Drawer is Up but no retracted or extended signal*)	
				bStepDone									:= TRUE;
			9: (*Drawer is retracted and Up*)		
				iSeqStep									:= 6; 
			10: (*Drawer is extended and Up*)		
				iSeqStep									:= 5; 	
			11, 12, 13, 14, 15: (*Error*)	
				_nErrorID									:= E_AlarmID.BothTIUExternRetractSignalDetected; 
				sMessage									:= 'Both Reed Switchs of Cylinder are Detected';
		END_CASE

///////////////////////////////////////////////////////////////////////////////////////////////////////////////////////////////////////////////////////////////////////////////
//	State: TBOT EAP checking, anticollision signal & drawer safe to move signal
///////////////////////////////////////////////////////////////////////////////////////////////////////////////////////////////////////////////////////////////////////////////				
	E_SeqSts.eTBotEAPSanityCheck:
		sMessage												:= ' Checking TBot EAP';
		_nErrorID												:= INT_TO_UDINT(M_IsEAPError(sMsg=>sMessage)) ;
		IF _nErrorID=0 THEN
			bStepDone											:= TRUE;
		END_IF

///////////////////////////////////////////////////////////////////////////////////////////////////////////////////////////////////////////////////////////////////////////////
//	State: Drawer Move Up OR Move Down
///////////////////////////////////////////////////////////////////////////////////////////////////////////////////////////////////////////////////////////////////////////////	
	E_SeqSts.eMoveDrawerUp, E_SeqSts.eMoveDrawerDown: //drawer up, drawer down
		sMessage												:= SEL(iStkSeqCase = E_SeqSts.eMoveDrawerUp,' Drawer Down',' Drawer Up');
		IF (NOT tUpDnlock) THEN
			tBef 												:= TIME();
			tUpDnlock											:= TRUE;
		END_IF
		iLibrySts[1]											:= M_nCmptUpDown(
																		bExtend		:= iStkSeqCase = E_SeqSts.eMoveDrawerUp,  
																		sErrorMSg	:= sMsg
																	);
		
		IF iLibrySts[1] = 10 THEN
			tAft												:= TIME();
			tUpDnlock											:= FALSE;
			sMessage											:= CONCAT(sMessage,'Duration: ');
			sMessage											:= CONCAT(sMessage,REAL_TO_STRING((TIME_TO_REAL(tAft-tBef)/1000)));
			sMessage											:= CONCAT(sMessage,' seconds');
			bStepDone											:= TRUE;
		ELSIF iLibrySts[1] = 99 THEN
			tUpDnlock											:= FALSE;
			sMessage											:= CONCAT(sMessage,sMsg);
			_bError												:= TRUE;
		END_IF
	
///////////////////////////////////////////////////////////////////////////////////////////////////////////////////////////////////////////////////////////////////////////////
//	State: Drawer Move In OR Move Out
///////////////////////////////////////////////////////////////////////////////////////////////////////////////////////////////////////////////////////////////////////////////			
	E_SeqSts.eMoveDrawerIn, E_SeqSts.eMoveDrawerOut: //drawer in, drawer out
		sMessage												:= SEL(iStkSeqCase = E_SeqSts.eMoveDrawerIn,
																	' Drawer Out',
																	' Drawer In');
		IF (NOT tInOutlock) THEN
			tBef 												:= TIME();
			tInOutlock											:= TRUE;
		END_IF	
		
		iLibrySts[1]											:= M_nCmptInOut(
																	bExtend			:= iStkSeqCase = E_SeqSts.eMoveDrawerOut,  
																	sErrorMSg		:= sMsg
																	);
		
		IF iLibrySts[1] = 10 THEN
			//<Cyl_Duration_Log>
				tAft											:= TIME();
				tInOutlock										:= FALSE;
				sMessage										:= CONCAT(sMessage,'Duration: ');
				sMessage										:= CONCAT(sMessage,REAL_TO_STRING((TIME_TO_REAL(tAft-tBef)/1000)));
				sMessage										:= CONCAT(sMessage,' seconds');
			//<Cyl_Duration_Log>
			bStepDone											:= TRUE;
			
		ELSIF iLibrySts[1] = 99 AND (bDebugCart AND stMLVIO.iAlarmCode = E_AlarmID.DrawerExtendError) THEN //to reset DwrExtError without stepping to process.E_SeqErr Step
			inTCDrawerExtRet.M_nOff();//inTCDrawerExtRet.M_nReset();
			iLibrySts[1]										:= 10;
			bStepDone											:= TRUE;
			
		ELSIF iLibrySts[1] = 99 THEN
			tInOutlock											:= FALSE;
			sMessage											:= CONCAT(sMessage,sMsg);
			_bError												:= TRUE;
		END_IF
		
///////////////////////////////////////////////////////////////////////////////////////////////////////////////////////////////////////////////////////////////////////////////
//	State: Turn OFF AP Air Valve (10Bar)	(Debug Cart only.)
///////////////////////////////////////////////////////////////////////////////////////////////////////////////////////////////////////////////////////////////////////////////
	E_SeqSts.eTurnOffAPAirValve: //only for debug cart front door
		sMessage												:= ' Turn Off AP Air Valve (10Bar)';
		stMLVIO.opAPAirSupplySol 								:= FALSE; //not able to false it maybe library turn it back on
		bStepDone												:= TRUE;
		
///////////////////////////////////////////////////////////////////////////////////////////////////////////////////////////////////////////////////////////////////////////////
//	State: Turn OFF Tester Air Valve (6Bar)	(Debug Cart only.)
///////////////////////////////////////////////////////////////////////////////////////////////////////////////////////////////////////////////////////////////////////////////		
	E_SeqSts.eTurnOffTesterAirValve: //only for debug cart front door
		sMessage												:= ' Turn Off Tester Air Valve (6Bar)';
		stMLVIO.opTesterDrawerAirSupplySol 						:= FALSE; //not able to false it maybe library turn it back on
		bStepDone												:= TRUE;
		
///////////////////////////////////////////////////////////////////////////////////////////////////////////////////////////////////////////////////////////////////////////////
//	State: Turn ON AP Air Valve (10Bar)	(Debug Cart only.)
///////////////////////////////////////////////////////////////////////////////////////////////////////////////////////////////////////////////////////////////////////////////
	E_SeqSts.eTurnOnAPAirValve: //only for debug cart front door
		IF bDebugCart THEN
			IF stMLVIO.ipAPPresentSensor THEN 
				sMessage										:= ' Turn on AP Air Valve (10Bar)';
				stMLVIO.opAPAirSupplySol						:= TRUE;
			END_IF
		END_IF
		
		bStepDone												:= TRUE;
	
///////////////////////////////////////////////////////////////////////////////////////////////////////////////////////////////////////////////////////////////////////////////
//	State: Turn ON Tesrer Air Valve (6Bar) (Debug Cart only.)
///////////////////////////////////////////////////////////////////////////////////////////////////////////////////////////////////////////////////////////////////////////////
	E_SeqSts.eTurnOnTesterAirValve: //only for debug cart front door
		IF bDebugCart THEN
			sMessage											:= ' Turn on Tester Air Valve (6Bar)';
			stMLVIO.opTesterDrawerAirSupplySol					:= TRUE;
		END_IF
		
		bStepDone												:= TRUE;
	
///////////////////////////////////////////////////////////////////////////////////////////////////////////////////////////////////////////////////////////////////////////////
//	State: On Drawer Extend Output only?? For what (Debug Cart only.)
///////////////////////////////////////////////////////////////////////////////////////////////////////////////////////////////////////////////////////////////////////////////
	E_SeqSts.eOnDrawerOutputOnly:
		inTCDrawerExtRet.M_nExtend(
			bExecute											:= TRUE);
		bStepDone												:= TRUE;
		
///////////////////////////////////////////////////////////////////////////////////////////////////////////////////////////////////////////////////////////////////////////////
//	State: Completed
///////////////////////////////////////////////////////////////////////////////////////////////////////////////////////////////////////////////////////////////////////////////		
	E_SeqSts.eDone:
		sMessage												:= ' Done';
		M_SequenceCommand										:= 10;
END_CASE	



//Checking any error, if error return, else continue next step
IF _nErrorID > 0 OR _bError THEN
	_bError													:= TRUE;
ELSIF (stMLVIO.bStep OR stMLVIO.bBypassSingleMove OR iStkSeqCase <= E_SeqSts.eSanityCheck) AND iStkSeqCase < E_SeqSts.eDone AND bStepDone THEN
	iSeqStep												:= iSeqStep + 1;
	stMLVIO.bStep											:= FALSE;
END_IF
END_METHOD

PROPERTY P_ErrClear : BOOL
GET
END_GET
SET
bErrClear 			:= P_ErrClear;
END_SET
END_PROPERTY

PROPERTY P_sEAPMessage : STRING
GET
//P_sEAPMessage:=sEAPMessage;
END_GET
END_PROPERTY

PROPERTY P_sMessage : string
GET
P_sMessage := sMessage;
END_GET
END_PROPERTY

PROPERTY PUBLIC P_stParam : ST_TCMultiLevelSeqParam
GET
P_stParam := stTCMLSeqParam;
END_GET
SET
stTCMLSeqParam := P_stParam;
END_SET
END_PROPERTY

PROPERTY PUBLIC P_stTCMultiLevelVIO : ST_TCMultiLevel_VIO
GET // PUBLIC
P_stTCMultiLevelVIO := stMLVIO;
END_GET
SET
stMLVIO := P_stTCMultiLevelVIO;
END_SET
END_PROPERTY

ACTION PermSD:
FC_BitToWord(
	BOOL_00		:= TRUE, 
	BOOL_01		:= TRUE, 
	BOOL_02		:= TRUE, 
	BOOL_03		:= TRUE, 
	BOOL_04		:= TRUE, 
	BOOL_05		:= TRUE, 
	BOOL_06		:= TRUE, 
	BOOL_07		:= TRUE, 
	BOOL_08		:= TRUE, 
	BOOL_09		:= TRUE, 
	BOOL_10		:= TRUE, 
	BOOL_11		:= TRUE, 
	BOOL_12		:= TRUE, 
	BOOL_13		:= TRUE, 
	BOOL_14		:= TRUE, 
	BOOL_15		:= TRUE, 
	Output_Word		=> TC_AP240Power_Perm);
	
FC_BitToWord(
	BOOL_00		:= FALSE, 
	BOOL_01		:= FALSE, 
	BOOL_02		:= FALSE, 
	BOOL_03		:= FALSE, 
	BOOL_04		:= FALSE, 
	BOOL_05		:= FALSE, 
	BOOL_06		:= FALSE, 
	BOOL_07		:= FALSE, 
	BOOL_08		:= FALSE, 
	BOOL_09		:= FALSE, 
	BOOL_10		:= FALSE, 
	BOOL_11		:= FALSE, 
	BOOL_12		:= FALSE, 
	BOOL_13		:= FALSE, 
	BOOL_14		:= FALSE, 
	BOOL_15		:= FALSE, 
	Output_Word		=> TC_AP240Power_SD);
END_ACTION

END_FUNCTION_BLOCK

(* stored: Version 1.1.0.1, ProductVersion 3.1.4022.18
   POU FB_TCMultiLevelSeq: Id {d05d5490-7299-4891-9098-6afe4d42641d}, SpecialFunc None
   Folder 1.LogicCyclic: Id {bce124f9-6199-4ae1-9f2b-c9842fd11f69}
   Folder 2.RemoteCommand: Id {4eb389e0-af3d-4110-8b0f-6611ef8c1085}
   Folder 3.Method: Id {9f15dea2-6fcc-41c2-a76e-822f05ed3928}
   Method AirOnOff: Id {125af07d-16d0-4314-bb0d-60a6457d3652}
   Method DwrAirOnInit: Id {345d20aa-8bac-429c-8166-21514382a04a}
   Method M_240APPwr: Id {158c9825-e25a-4c2e-b234-be6bf1c15da6}
   Method M_240TstPwr: Id {3f386753-5c64-4d66-9d59-10a613bee6e1}
   Method M_AboveLeakageChecking: Id {275d87db-42a5-495e-bfda-c82567e8de61}
   Method M_APSanityCheck: Id {09eea1b5-4824-425a-98ec-d047b3c77afc}
   Method M_GetTIUStatus: Id {fb2f011d-463a-4a71-89d1-e39639a1bcb2}
   Method M_InitializeCommand: Id {942afd54-b1c1-4798-a25e-93d4e56947c9}
   Method M_InputBackDoor: Id {671b77c7-1523-4320-b84b-a1aa06230f8a}
   Method M_InterlockTII: Id {88edcd8a-14ef-48d8-99bb-1f383da7f5f2}
   Method M_IOMapping: Id {e3ee4a20-fc21-496d-a3bf-b8671140ad85}
   Method M_IsEAPError: Id {e48d78cc-04e2-4730-bd22-ba4cf04a5d13}
   Method M_nCmptInOut: Id {c3fa4dbd-caf3-402c-9f5c-8537b02d385b}
   Method M_nCmptUpDown: Id {5d35f409-d04b-4a9c-b96e-73bd2f3eaefb}
   Method M_nCyclic: Id {d892c72f-d562-4499-959e-3dade4011a0e}
   Method M_nDPSPowerOnOff: Id {23018554-f366-4756-8a3f-c3b4774f229e}
   Method M_Pwr: Id {b22dc467-cf02-4b3c-a883-1f42dfbedd64}
   Method M_RemoteSecondary24VPowerOnOff: Id {5b27ece6-923e-4133-9791-5ed0b8c18038}
   Method M_Secondary24VPower: Id {3e6ef57f-d508-4f74-9216-2c66b14c555c}
   Method M_SeqAlmRset: Id {5b34250c-a5b5-4e02-9baa-75a97529b213}
   Method M_SequenceCommand: Id {678f1901-d1d0-4ab8-9f2a-61ea8068b3b1}
   Property P_ErrClear: Id {71cdd4bd-ba6b-49c4-b14e-5c7fbe82818d}
   Get Get: Id {0807d10a-eeb3-4695-8e30-917d319f4063}
   Set Set: Id {310d3e4b-5140-4768-8917-acf05dd9b656}
   Property P_sEAPMessage: Id {18ba7c01-66e5-4c94-b5ad-aff18d302282}
   Get Get: Id {27fb4b6d-0ca2-4d6f-8e3d-004883171bad}
   Property P_sMessage: Id {dc9296a0-98ab-4663-8d36-692691155897}
   Get Get: Id {a4fb15c2-10b8-4edb-bb87-4f4e0e50a2a6}
   Property P_stParam: Id {265f886d-b4db-434b-ba25-4d3682189875}
   Get Get: Id {169fc1e3-c53d-48e4-8a95-0c7e2cfbff75}
   Set Set: Id {06c4b386-8ad2-4d1e-8d4a-b037f883ddcd}
   Property P_stTCMultiLevelVIO: Id {b9b49ce6-01ea-4b6a-ba50-0e5aa0c680b0}
   Get Get: Id {d386f3a9-6214-4e5f-82b6-219668a4713d}
   Set Set: Id {fe6c83cd-158b-4b53-ba82-75a689b4212b}
   Action PermSD: Id {8f6317db-aed8-42b3-a3e7-277a2f515be4} *)
